LIN {X 0,Y 474.638,Z 146.861,A -85,B 0,C 180,E1 -7446.642,E2 -7446.642} C_VEL
LIN {X 0,Y 474.676,Z 147.003,A -85,B 0,C 180,E1 -7448.104,E2 -7448.104} C_VEL
LIN {X 0,Y 475.943,Z 154.468,A -85,B 0,C 180,E1 -7449.695,E2 -7449.695} C_VEL
LIN {X 0,Y 475.766,Z 161.873,A -85,B 0,C 180,E1 -7451.18,E2 -7451.18} C_VEL
LIN {X 0,Y 475.04,Z 165.15,A -85,B 0,C 180,E1 -7451.743,E2 -7451.743} C_VEL
LIN {X 0,Y 472.97,Z 170.29,A -85,B 0,C 180,E1 -7452.392,E2 -7452.392} C_VEL
LIN {X 0,Y 471.001,Z 176.225,A -85,B 0,C 180,E1 -7452.91,E2 -7452.91} C_VEL
LIN {X 0,Y 470.387,Z 181.246,A -85,B 0,C 180,E1 -7453.195,E2 -7453.195} C_VEL
LIN {X 0,Y 470.756,Z 184.775,A -85,B 0,C 180,E1 -7453.315,E2 -7453.315} C_VEL
LIN {X 0,Y 471.43,Z 190.109,A -85,B 0,C 180,E1 -7453.423,E2 -7453.423} C_VEL
LIN {X 0,Y 470.672,Z 280.468,A -85,B 0,C 180,E1 -7454.825,E2 -7454.825} C_VEL
LIN {X 0,Y 470.313,Z 294.355,A -85,B 0,C 180,E1 -7455.228,E2 -7455.228} C_VEL
LIN {X 0,Y 469.955,Z 306.775,A -85,B 0,C 180,E1 -7455.77,E2 -7455.77} C_VEL
LIN {X 0,Y 469.52,Z 318.965,A -85,B 0,C 180,E1 -7456.497,E2 -7456.497} C_VEL
LIN {X 0,Y 469.081,Z 330.013,A -85,B 0,C 180,E1 -7457.343,E2 -7457.343} C_VEL
LIN {X 0,Y 468.559,Z 340.263,A -85,B 0,C 180,E1 -7458.317,E2 -7458.317} C_VEL
LIN {X 0,Y 468.098,Z 349.46,A -85,B 0,C 180,E1 -7459.402,E2 -7459.402} C_VEL
LIN {X 0,Y 467.642,Z 358.386,A -85,B 0,C 180,E1 -7460.703,E2 -7460.703} C_VEL
LIN {X 0,Y 467.255,Z 365.574,A -85,B 0,C 180,E1 -7462.003,E2 -7462.003} C_VEL
LIN {X 0,Y 467.028,Z 371.353,A -85,B 0,C 180,E1 -7463.313,E2 -7463.313} C_VEL
LIN {X 0,Y 466.805,Z 376.452,A -85,B 0,C 180,E1 -7464.817,E2 -7464.817} C_VEL
LIN {X 0,Y 466.751,Z 378.743,A -85,B 0,C 180,E1 -7465.682,E2 -7465.682} C_VEL
LIN {X 0,Y 466.79,Z 380.605,A -85,B 0,C 180,E1 -7466.547,E2 -7466.547} C_VEL
LIN {X 0,Y 466.693,Z 382.013,A -85,B 0,C 180,E1 -7467.411,E2 -7467.411} C_VEL
LIN {X 0,Y 466.621,Z 383.629,A -85,B 0,C 180,E1 -7469.137,E2 -7469.137} C_VEL
LIN {X 0,Y 466.601,Z 383.866,A -85,B 0,C 180,E1 -7470,E2 -7470} C_VEL
LIN {X 0,Y 466.621,Z 383.68,A -85,B 0,C 180,E1 -7470.863,E2 -7470.863} C_VEL
LIN {X 0,Y 466.693,Z 382.129,A -85,B 0,C 180,E1 -7472.589,E2 -7472.589} C_VEL
LIN {X 0,Y 466.788,Z 380.771,A -85,B 0,C 180,E1 -7473.453,E2 -7473.453} C_VEL
LIN {X 0,Y 466.736,Z 377.908,A -85,B 0,C 180,E1 -7474.75,E2 -7474.75} C_VEL
LIN {X 0,Y 466.975,Z 374.018,A -85,B 0,C 180,E1 -7476.047,E2 -7476.047} C_VEL
LIN {X 0,Y 467.1,Z 369.005,A -85,B 0,C 180,E1 -7477.348,E2 -7477.348} C_VEL
LIN {X 0,Y 467.381,Z 362.693,A -85,B 0,C 180,E1 -7478.648,E2 -7478.648} C_VEL
LIN {X 0,Y 467.761,Z 354.79,A -85,B 0,C 180,E1 -7479.95,E2 -7479.95} C_VEL
LIN {X 0,Y 468.291,Z 344.958,A -85,B 0,C 180,E1 -7481.251,E2 -7481.251} C_VEL
LIN {X 0,Y 468.868,Z 334.644,A -85,B 0,C 180,E1 -7482.333,E2 -7482.333} C_VEL
LIN {X 0,Y 469.315,Z 323.077,A -85,B 0,C 180,E1 -7483.306,E2 -7483.306} C_VEL
LIN {X 0,Y 469.774,Z 311.433,A -85,B 0,C 180,E1 -7484.07,E2 -7484.07} C_VEL
LIN {X 0,Y 470.257,Z 299.391,A -85,B 0,C 180,E1 -7484.663,E2 -7484.663} C_VEL
LIN {X 0,Y 470.544,Z 286.28,A -85,B 0,C 180,E1 -7485.124,E2 -7485.124} C_VEL
LIN {X 0,Y 470.782,Z 273.664,A -85,B 0,C 180,E1 -7485.393,E2 -7485.393} C_VEL
LIN {X 0,Y 471.364,Z 188.194,A -85,B 0,C 180,E1 -7486.702,E2 -7486.702} C_VEL
LIN {X 0,Y 468.444,Z 172.801,A -85,B 0,C 180,E1 -7487.059,E2 -7487.059} C_VEL
LIN {X 0,Y 469,Z 157.256,A -85,B 0,C 180,E1 -7490.161,E2 -7490.161} C_VEL
LIN {X 0,Y 468.247,Z 151.065,A -85,B 0,C 180,E1 -7491.476,E2 -7491.476} C_VEL
LIN {X 0,Y 467.603,Z 147.741,A -85,B 0,C 180,E1 -7492.245,E2 -7492.245} C_VEL
LIN {X 0,Y 467.616,Z 147.734,A -85,B 0,C 180,E1 -7495.608,E2 -7495.608} C_VEL
LIN {X 0,Y 467.622,Z 147.732,A -85,B 0,C 180,E1 -7497.769,E2 -7497.769} C_VEL
LIN {X 0,Y 467.569,Z 147.741,A -85,B 0,C 180,E1 -7501.044,E2 -7501.044} C_VEL
LIN {X 0,Y 467.578,Z 147.741,A -85,B 0,C 180,E1 -7504.24,E2 -7504.24} C_VEL
LIN {X 0,Y 467.549,Z 147.741,A -85,B 0,C 180,E1 -7507.186,E2 -7507.186} C_VEL
LIN {X 0,Y 467.575,Z 147.745,A -85,B 0,C 180,E1 -7510.265,E2 -7510.265} C_VEL
LIN {X 0,Y 467.587,Z 147.74,A -85,B 0,C 180,E1 -7512.567,E2 -7512.567} C_VEL
LIN {X 0,Y 467.571,Z 147.738,A -85,B 0,C 180,E1 -7515.053,E2 -7515.053} C_VEL
LIN {X 0,Y 467.589,Z 147.736,A -85,B 0,C 180,E1 -7517.44,E2 -7517.44} C_VEL
LIN {X 0,Y 467.583,Z 147.737,A -85,B 0,C 180,E1 -7520.855,E2 -7520.855} C_VEL
LIN {X 0,Y 467.559,Z 147.743,A -85,B 0,C 180,E1 -7524.261,E2 -7524.261} C_VEL
LIN {X 0,Y 467.582,Z 147.739,A -85,B 0,C 180,E1 -7527.321,E2 -7527.321} C_VEL
LIN {X 0,Y 467.569,Z 147.738,A -85,B 0,C 180,E1 -7530.667,E2 -7530.667} C_VEL
LIN {X 0,Y 467.616,Z 147.735,A -85,B 0,C 180,E1 -7533.2,E2 -7533.2} C_VEL
LIN {X 0,Y 467.592,Z 147.735,A -85,B 0,C 180,E1 -7536.468,E2 -7536.468} C_VEL
LIN {X 0,Y 467.624,Z 147.735,A -85,B 0,C 180,E1 -7539.777,E2 -7539.777} C_VEL
LIN {X 0,Y 467.608,Z 147.733,A -85,B 0,C 180,E1 -7542.507,E2 -7542.507} C_VEL
LIN {X 0,Y 467.606,Z 147.741,A -85,B 0,C 180,E1 -7545.196,E2 -7545.196} C_VEL
LIN {X 0,Y 467.655,Z 147.728,A -85,B 0,C 180,E1 -7547.854,E2 -7547.854} C_VEL
LIN {X 0,Y 467.681,Z 147.729,A -85,B 0,C 180,E1 -7551.357,E2 -7551.357} C_VEL
LIN {X 0,Y 467.734,Z 147.718,A -85,B 0,C 180,E1 -7553.962,E2 -7553.962} C_VEL
LIN {X 0,Y 467.859,Z 147.704,A -85,B 0,C 180,E1 -7557.417,E2 -7557.417} C_VEL
LIN {X 0,Y 467.881,Z 147.699,A -85,B 0,C 180,E1 -7560,E2 -7560} C_VEL
LIN {X 0,Y 467.858,Z 147.708,A -85,B 0,C 180,E1 -7562.583,E2 -7562.583} C_VEL
LIN {X 0,Y 467.735,Z 147.719,A -85,B 0,C 180,E1 -7566.037,E2 -7566.037} C_VEL
LIN {X 0,Y 467.679,Z 147.731,A -85,B 0,C 180,E1 -7568.643,E2 -7568.643} C_VEL
LIN {X 0,Y 467.655,Z 147.731,A -85,B 0,C 180,E1 -7572.145,E2 -7572.145} C_VEL
LIN {X 0,Y 467.638,Z 147.731,A -85,B 0,C 180,E1 -7575.695,E2 -7575.695} C_VEL
LIN {X 0,Y 467.621,Z 147.732,A -85,B 0,C 180,E1 -7579.308,E2 -7579.308} C_VEL
LIN {X 0,Y 467.534,Z 147.75,A -85,B 0,C 180,E1 -7582.074,E2 -7582.074} C_VEL
LIN {X 0,Y 467.583,Z 147.737,A -85,B 0,C 180,E1 -7584.889,E2 -7584.889} C_VEL
LIN {X 0,Y 467.618,Z 147.737,A -85,B 0,C 180,E1 -7587.769,E2 -7587.769} C_VEL
LIN {X 0,Y 467.567,Z 147.739,A -85,B 0,C 180,E1 -7591.045,E2 -7591.045} C_VEL
LIN {X 0,Y 467.587,Z 147.738,A -85,B 0,C 180,E1 -7594.242,E2 -7594.242} C_VEL
LIN {X 0,Y 467.542,Z 147.744,A -85,B 0,C 180,E1 -7597.186,E2 -7597.186} C_VEL
LIN {X 0,Y 467.57,Z 147.739,A -85,B 0,C 180,E1 -7600.266,E2 -7600.266} C_VEL
LIN {X 0,Y 467.548,Z 147.745,A -85,B 0,C 180,E1 -7603.745,E2 -7603.745} C_VEL
LIN {X 0,Y 467.548,Z 147.741,A -85,B 0,C 180,E1 -7606.255,E2 -7606.255} C_VEL
LIN {X 0,Y 467.567,Z 147.74,A -85,B 0,C 180,E1 -7608.725,E2 -7608.725} C_VEL
LIN {X 0,Y 467.564,Z 147.739,A -85,B 0,C 180,E1 -7611.956,E2 -7611.956} C_VEL
LIN {X 0,Y 467.559,Z 147.747,A -85,B 0,C 180,E1 -7615.167,E2 -7615.167} C_VEL
LIN {X 0,Y 467.581,Z 147.737,A -85,B 0,C 180,E1 -7618.26,E2 -7618.26} C_VEL
LIN {X 0,Y 467.545,Z 147.745,A -85,B 0,C 180,E1 -7621.248,E2 -7621.248} C_VEL
LIN {X 0,Y 467.592,Z 147.743,A -85,B 0,C 180,E1 -7624.494,E2 -7624.494} C_VEL
LIN {X 0,Y 467.598,Z 147.812,A -85,B 0,C 180,E1 -7624.643,E2 -7624.643} C_VEL
LIN {X 0,Y 469.719,Z 159.111,A -85,B 0,C 180,E1 -7626.874,E2 -7626.874} C_VEL
LIN {X 0,Y 469.057,Z 174.117,A -85,B 0,C 180,E1 -7629.613,E2 -7629.613} C_VEL
LIN {X 0,Y 468.416,Z 190.342,A -85,B 0,C 180,E1 -7632.538,E2 -7632.538} C_VEL
LIN {X 0,Y 468.346,Z 192.794,A -85,B 0,C 180,E1 -7632.978,E2 -7632.978} C_VEL
LIN {X 0,Y 471.213,Z 210.729,A -85,B 0,C 180,E1 -7633.367,E2 -7633.367} C_VEL
LIN {X 0,Y 470.577,Z 300.893,A -85,B 0,C 180,E1 -7634.766,E2 -7634.766} C_VEL
LIN {X 0,Y 470.209,Z 314.155,A -85,B 0,C 180,E1 -7635.142,E2 -7635.142} C_VEL
LIN {X 0,Y 469.778,Z 326.312,A -85,B 0,C 180,E1 -7635.654,E2 -7635.654} C_VEL
LIN {X 0,Y 469.262,Z 338.578,A -85,B 0,C 180,E1 -7636.356,E2 -7636.356} C_VEL
LIN {X 0,Y 468.763,Z 350.191,A -85,B 0,C 180,E1 -7637.226,E2 -7637.226} C_VEL
LIN {X 0,Y 468.251,Z 360.609,A -85,B 0,C 180,E1 -7638.2,E2 -7638.2} C_VEL
LIN {X 0,Y 467.794,Z 369.142,A -85,B 0,C 180,E1 -7639.176,E2 -7639.176} C_VEL
LIN {X 0,Y 467.46,Z 377.017,A -85,B 0,C 180,E1 -7640.262,E2 -7640.262} C_VEL
LIN {X 0,Y 467.108,Z 384.706,A -85,B 0,C 180,E1 -7641.565,E2 -7641.565} C_VEL
LIN {X 0,Y 466.853,Z 391.796,A -85,B 0,C 180,E1 -7643.083,E2 -7643.083} C_VEL
LIN {X 0,Y 466.762,Z 396.513,A -85,B 0,C 180,E1 -7644.384,E2 -7644.384} C_VEL
LIN {X 0,Y 466.645,Z 400.115,A -85,B 0,C 180,E1 -7645.681,E2 -7645.681} C_VEL
LIN {X 0,Y 466.66,Z 401.975,A -85,B 0,C 180,E1 -7646.546,E2 -7646.546} C_VEL
LIN {X 0,Y 466.66,Z 403.369,A -85,B 0,C 180,E1 -7647.411,E2 -7647.411} C_VEL
LIN {X 0,Y 466.59,Z 404.969,A -85,B 0,C 180,E1 -7649.137,E2 -7649.137} C_VEL
LIN {X 0,Y 466.6,Z 405.185,A -85,B 0,C 180,E1 -7650,E2 -7650} C_VEL
LIN {X 0,Y 466.607,Z 404.363,A -85,B 0,C 180,E1 -7651.726,E2 -7651.726} C_VEL
LIN {X 0,Y 466.66,Z 403.37,A -85,B 0,C 180,E1 -7652.59,E2 -7652.59} C_VEL
LIN {X 0,Y 466.66,Z 401.976,A -85,B 0,C 180,E1 -7653.454,E2 -7653.454} C_VEL
LIN {X 0,Y 466.688,Z 399.044,A -85,B 0,C 180,E1 -7654.751,E2 -7654.751} C_VEL
LIN {X 0,Y 466.753,Z 395.074,A -85,B 0,C 180,E1 -7656.05,E2 -7656.05} C_VEL
LIN {X 0,Y 466.944,Z 388.971,A -85,B 0,C 180,E1 -7657.568,E2 -7657.568} C_VEL
LIN {X 0,Y 467.215,Z 382.3,A -85,B 0,C 180,E1 -7658.869,E2 -7658.869} C_VEL
LIN {X 0,Y 467.578,Z 374.024,A -85,B 0,C 180,E1 -7660.172,E2 -7660.172} C_VEL
LIN {X 0,Y 468.022,Z 365.541,A -85,B 0,C 180,E1 -7661.257,E2 -7661.257} C_VEL
LIN {X 0,Y 468.58,Z 355.481,A -85,B 0,C 180,E1 -7662.302,E2 -7662.302} C_VEL
LIN {X 0,Y 468.966,Z 344.686,A -85,B 0,C 180,E1 -7663.211,E2 -7663.211} C_VEL
LIN {X 0,Y 469.487,Z 333.316,A -85,B 0,C 180,E1 -7663.968,E2 -7663.968} C_VEL
LIN {X 0,Y 469.968,Z 321.649,A -85,B 0,C 180,E1 -7664.561,E2 -7664.561} C_VEL
LIN {X 0,Y 470.351,Z 310.034,A -85,B 0,C 180,E1 -7664.992,E2 -7664.992} C_VEL
LIN {X 0,Y 470.631,Z 296.424,A -85,B 0,C 180,E1 -7665.315,E2 -7665.315} C_VEL
LIN {X 0,Y 471.101,Z 210.051,A -85,B 0,C 180,E1 -7666.645,E2 -7666.645} C_VEL
LIN {X 0,Y 468.324,Z 192.816,A -85,B 0,C 180,E1 -7667.016,E2 -7667.016} C_VEL
LIN {X 0,Y 468.935,Z 176.595,A -85,B 0,C 180,E1 -7669.935,E2 -7669.935} C_VEL
LIN {X 0,Y 469.569,Z 162.843,A -85,B 0,C 180,E1 -7672.436,E2 -7672.436} C_VEL
LIN {X 0,Y 469.566,Z 157.831,A -85,B 0,C 180,E1 -7673.367,E2 -7673.367} C_VEL
LIN {X 0,Y 467.586,Z 147.743,A -85,B 0,C 180,E1 -7675.407,E2 -7675.407} C_VEL
LIN {X 0,Y 467.545,Z 147.743,A -85,B 0,C 180,E1 -7678.752,E2 -7678.752} C_VEL
LIN {X 0,Y 467.559,Z 147.74,A -85,B 0,C 180,E1 -7681.742,E2 -7681.742} C_VEL
LIN {X 0,Y 467.559,Z 147.747,A -85,B 0,C 180,E1 -7684.833,E2 -7684.833} C_VEL
LIN {X 0,Y 467.564,Z 147.739,A -85,B 0,C 180,E1 -7688.044,E2 -7688.044} C_VEL
LIN {X 0,Y 467.567,Z 147.739,A -85,B 0,C 180,E1 -7691.404,E2 -7691.404} C_VEL
LIN {X 0,Y 467.565,Z 147.742,A -85,B 0,C 180,E1 -7694.947,E2 -7694.947} C_VEL
LIN {X 0,Y 467.573,Z 147.744,A -85,B 0,C 180,E1 -7698.597,E2 -7698.597} C_VEL
LIN {X 0,Y 467.562,Z 147.742,A -85,B 0,C 180,E1 -7701.955,E2 -7701.955} C_VEL
LIN {X 0,Y 467.562,Z 147.739,A -85,B 0,C 180,E1 -7705.167,E2 -7705.167} C_VEL
LIN {X 0,Y 467.582,Z 147.744,A -85,B 0,C 180,E1 -7708.26,E2 -7708.26} C_VEL
LIN {X 0,Y 467.555,Z 147.74,A -85,B 0,C 180,E1 -7711.249,E2 -7711.249} C_VEL
LIN {X 0,Y 467.584,Z 147.742,A -85,B 0,C 180,E1 -7714.158,E2 -7714.158} C_VEL
LIN {X 0,Y 467.575,Z 147.737,A -85,B 0,C 180,E1 -7716.996,E2 -7716.996} C_VEL
LIN {X 0,Y 467.622,Z 147.739,A -85,B 0,C 180,E1 -7719.777,E2 -7719.777} C_VEL
LIN {X 0,Y 467.597,Z 147.735,A -85,B 0,C 180,E1 -7722.506,E2 -7722.506} C_VEL
LIN {X 0,Y 467.606,Z 147.736,A -85,B 0,C 180,E1 -7725.196,E2 -7725.196} C_VEL
LIN {X 0,Y 467.656,Z 147.732,A -85,B 0,C 180,E1 -7727.855,E2 -7727.855} C_VEL
LIN {X 0,Y 467.68,Z 147.731,A -85,B 0,C 180,E1 -7731.357,E2 -7731.357} C_VEL
LIN {X 0,Y 467.735,Z 147.719,A -85,B 0,C 180,E1 -7733.963,E2 -7733.963} C_VEL
LIN {X 0,Y 467.859,Z 147.709,A -85,B 0,C 180,E1 -7737.417,E2 -7737.417} C_VEL
LIN {X 0,Y 467.882,Z 147.7,A -85,B 0,C 180,E1 -7740,E2 -7740} C_VEL
LIN {X 0,Y 467.859,Z 147.703,A -85,B 0,C 180,E1 -7742.583,E2 -7742.583} C_VEL
LIN {X 0,Y 467.724,Z 147.719,A -85,B 0,C 180,E1 -7746.038,E2 -7746.038} C_VEL
LIN {X 0,Y 467.68,Z 147.728,A -85,B 0,C 180,E1 -7748.643,E2 -7748.643} C_VEL
LIN {X 0,Y 467.656,Z 147.728,A -85,B 0,C 180,E1 -7752.146,E2 -7752.146} C_VEL
LIN {X 0,Y 467.639,Z 147.729,A -85,B 0,C 180,E1 -7755.695,E2 -7755.695} C_VEL
LIN {X 0,Y 467.618,Z 147.739,A -85,B 0,C 180,E1 -7758.765,E2 -7758.765} C_VEL
LIN {X 0,Y 467.58,Z 147.738,A -85,B 0,C 180,E1 -7761.268,E2 -7761.268} C_VEL
LIN {X 0,Y 467.572,Z 147.739,A -85,B 0,C 180,E1 -7763.943,E2 -7763.943} C_VEL
LIN {X 0,Y 467.617,Z 147.735,A -85,B 0,C 180,E1 -7766.8,E2 -7766.8} C_VEL
LIN {X 0,Y 467.554,Z 147.741,A -85,B 0,C 180,E1 -7769.738,E2 -7769.738} C_VEL
LIN {X 0,Y 467.584,Z 147.738,A -85,B 0,C 180,E1 -7772.759,E2 -7772.759} C_VEL
LIN {X 0,Y 467.554,Z 147.744,A -85,B 0,C 180,E1 -7775.89,E2 -7775.89} C_VEL
LIN {X 0,Y 467.583,Z 147.736,A -85,B 0,C 180,E1 -7779.145,E2 -7779.145} C_VEL
LIN {X 0,Y 467.587,Z 147.737,A -85,B 0,C 180,E1 -7782.567,E2 -7782.567} C_VEL
LIN {X 0,Y 467.571,Z 147.738,A -85,B 0,C 180,E1 -7785.053,E2 -7785.053} C_VEL
LIN {X 0,Y 467.59,Z 147.739,A -85,B 0,C 180,E1 -7787.44,E2 -7787.44} C_VEL
LIN {X 0,Y 467.561,Z 147.739,A -85,B 0,C 180,E1 -7790.853,E2 -7790.853} C_VEL
LIN {X 0,Y 467.56,Z 147.74,A -85,B 0,C 180,E1 -7794.261,E2 -7794.261} C_VEL
LIN {X 0,Y 467.581,Z 147.742,A -85,B 0,C 180,E1 -7797.322,E2 -7797.322} C_VEL
LIN {X 0,Y 467.571,Z 147.738,A -85,B 0,C 180,E1 -7800.668,E2 -7800.668} C_VEL
LIN {X 0,Y 467.619,Z 147.738,A -85,B 0,C 180,E1 -7803.2,E2 -7803.2} C_VEL
LIN {X 0,Y 467.595,Z 147.738,A -85,B 0,C 180,E1 -7806.468,E2 -7806.468} C_VEL
LIN {X 0,Y 467.632,Z 147.918,A -85,B 0,C 180,E1 -7807.931,E2 -7807.931} C_VEL
LIN {X 0,Y 468.992,Z 155.682,A -85,B 0,C 180,E1 -7809.61,E2 -7809.61} C_VEL
LIN {X 0,Y 468.564,Z 169.167,A -85,B 0,C 180,E1 -7812.318,E2 -7812.318} C_VEL
LIN {X 0,Y 468.434,Z 172.751,A -85,B 0,C 180,E1 -7813.024,E2 -7813.024} C_VEL
LIN {X 0,Y 470.756,Z 184.775,A -85,B 0,C 180,E1 -7813.315,E2 -7813.315} C_VEL
LIN {X 0,Y 470.8,Z 187.997,A -85,B 0,C 180,E1 -7813.367,E2 -7813.367} C_VEL
LIN {X 0,Y 469.376,Z 192.433,A -85,B 0,C 180,E1 -7813.384,E2 -7813.384} C_VEL
LIN {X 0,Y 465.208,Z 201.121,A -85,B 0,C 180,E1 -7813.366,E2 -7813.366} C_VEL
LIN {X 0,Y 464.48,Z 205.116,A -85,B 0,C 180,E1 -7813.402,E2 -7813.402} C_VEL
LIN {X 0,Y 463.829,Z 280.648,A -85,B 0,C 180,E1 -7814.595,E2 -7814.595} C_VEL
LIN {X 0,Y 463.469,Z 294.528,A -85,B 0,C 180,E1 -7815.005,E2 -7815.005} C_VEL
LIN {X 0,Y 463.083,Z 306.945,A -85,B 0,C 180,E1 -7815.554,E2 -7815.554} C_VEL
LIN {X 0,Y 462.643,Z 318.812,A -85,B 0,C 180,E1 -7816.27,E2 -7816.27} C_VEL
LIN {X 0,Y 462.175,Z 328.894,A -85,B 0,C 180,E1 -7817.039,E2 -7817.039} C_VEL
LIN {X 0,Y 461.655,Z 339.368,A -85,B 0,C 180,E1 -7818.029,E2 -7818.029} C_VEL
LIN {X 0,Y 461.162,Z 347.927,A -85,B 0,C 180,E1 -7819.018,E2 -7819.018} C_VEL
LIN {X 0,Y 460.746,Z 355.81,A -85,B 0,C 180,E1 -7820.119,E2 -7820.119} C_VEL
LIN {X 0,Y 460.315,Z 363.517,A -85,B 0,C 180,E1 -7821.439,E2 -7821.439} C_VEL
LIN {X 0,Y 460.001,Z 370.587,A -85,B 0,C 180,E1 -7822.979,E2 -7822.979} C_VEL
LIN {X 0,Y 459.87,Z 375.297,A -85,B 0,C 180,E1 -7824.299,E2 -7824.299} C_VEL
LIN {X 0,Y 459.658,Z 378.906,A -85,B 0,C 180,E1 -7825.616,E2 -7825.616} C_VEL
LIN {X 0,Y 459.701,Z 380.769,A -85,B 0,C 180,E1 -7826.494,E2 -7826.494} C_VEL
LIN {X 0,Y 459.617,Z 382.175,A -85,B 0,C 180,E1 -7827.371,E2 -7827.371} C_VEL
LIN {X 0,Y 459.525,Z 383.792,A -85,B 0,C 180,E1 -7829.124,E2 -7829.124} C_VEL
LIN {X 0,Y 459.504,Z 384.028,A -85,B 0,C 180,E1 -7830,E2 -7830} C_VEL
LIN {X 0,Y 459.525,Z 383.841,A -85,B 0,C 180,E1 -7830.876,E2 -7830.876} C_VEL
LIN {X 0,Y 459.617,Z 382.29,A -85,B 0,C 180,E1 -7832.629,E2 -7832.629} C_VEL
LIN {X 0,Y 459.699,Z 380.933,A -85,B 0,C 180,E1 -7833.506,E2 -7833.506} C_VEL
LIN {X 0,Y 459.664,Z 378.069,A -85,B 0,C 180,E1 -7834.824,E2 -7834.824} C_VEL
LIN {X 0,Y 459.912,Z 374.179,A -85,B 0,C 180,E1 -7836.141,E2 -7836.141} C_VEL
LIN {X 0,Y 460.05,Z 369.165,A -85,B 0,C 180,E1 -7837.461,E2 -7837.461} C_VEL
LIN {X 0,Y 460.361,Z 362.853,A -85,B 0,C 180,E1 -7838.781,E2 -7838.781} C_VEL
LIN {X 0,Y 460.744,Z 354.95,A -85,B 0,C 180,E1 -7840.103,E2 -7840.103} C_VEL
LIN {X 0,Y 461.34,Z 345.116,A -85,B 0,C 180,E1 -7841.422,E2 -7841.422} C_VEL
LIN {X 0,Y 461.93,Z 334.801,A -85,B 0,C 180,E1 -7842.521,E2 -7842.521} C_VEL
LIN {X 0,Y 462.382,Z 323.681,A -85,B 0,C 180,E1 -7843.474,E2 -7843.474} C_VEL
LIN {X 0,Y 462.908,Z 311.587,A -85,B 0,C 180,E1 -7844.283,E2 -7844.283} C_VEL
LIN {X 0,Y 463.387,Z 299.543,A -85,B 0,C 180,E1 -7844.885,E2 -7844.885} C_VEL
LIN {X 0,Y 463.694,Z 286.428,A -85,B 0,C 180,E1 -7845.353,E2 -7845.353} C_VEL
LIN {X 0,Y 463.943,Z 273.798,A -85,B 0,C 180,E1 -7845.626,E2 -7845.626} C_VEL
LIN {X 0,Y 464.469,Z 188.389,A -85,B 0,C 180,E1 -7846.956,E2 -7846.956} C_VEL
LIN {X 0,Y 461.514,Z 172.908,A -85,B 0,C 180,E1 -7847.332,E2 -7847.332} C_VEL
LIN {X 0,Y 462.052,Z 158.489,A -85,B 0,C 180,E1 -7850.245,E2 -7850.245} C_VEL
LIN {X 0,Y 461.404,Z 152.909,A -85,B 0,C 180,E1 -7851.442,E2 -7851.442} C_VEL
LIN {X 0,Y 460.568,Z 148.617,A -85,B 0,C 180,E1 -7852.426,E2 -7852.426} C_VEL
LIN {X 0,Y 460.57,Z 148.612,A -85,B 0,C 180,E1 -7855.802,E2 -7855.802} C_VEL
LIN {X 0,Y 460.554,Z 148.614,A -85,B 0,C 180,E1 -7858.233,E2 -7858.233} C_VEL
LIN {X 0,Y 460.522,Z 148.617,A -85,B 0,C 180,E1 -7861.282,E2 -7861.282} C_VEL
LIN {X 0,Y 460.524,Z 148.624,A -85,B 0,C 180,E1 -7864.504,E2 -7864.504} C_VEL
LIN {X 0,Y 460.502,Z 148.619,A -85,B 0,C 180,E1 -7867.623,E2 -7867.623} C_VEL
LIN {X 0,Y 460.54,Z 148.621,A -85,B 0,C 180,E1 -7870.269,E2 -7870.269} C_VEL
LIN {X 0,Y 460.501,Z 148.619,A -85,B 0,C 180,E1 -7873.375,E2 -7873.375} C_VEL
LIN {X 0,Y 460.5,Z 148.621,A -85,B 0,C 180,E1 -7876.624,E2 -7876.624} C_VEL
LIN {X 0,Y 460.542,Z 148.617,A -85,B 0,C 180,E1 -7879.73,E2 -7879.73} C_VEL
LIN {X 0,Y 460.5,Z 148.62,A -85,B 0,C 180,E1 -7882.524,E2 -7882.524} C_VEL
LIN {X 0,Y 460.546,Z 148.618,A -85,B 0,C 180,E1 -7885.624,E2 -7885.624} C_VEL
LIN {X 0,Y 460.537,Z 148.614,A -85,B 0,C 180,E1 -7888.744,E2 -7888.744} C_VEL
LIN {X 0,Y 460.581,Z 148.61,A -85,B 0,C 180,E1 -7892.254,E2 -7892.254} C_VEL
LIN {X 0,Y 460.558,Z 148.612,A -85,B 0,C 180,E1 -7894.705,E2 -7894.705} C_VEL
LIN {X 0,Y 460.51,Z 148.625,A -85,B 0,C 180,E1 -7897.571,E2 -7897.571} C_VEL
LIN {X 0,Y 460.569,Z 148.61,A -85,B 0,C 180,E1 -7900.384,E2 -7900.384} C_VEL
LIN {X 0,Y 460.565,Z 148.616,A -85,B 0,C 180,E1 -7903.146,E2 -7903.146} C_VEL
LIN {X 0,Y 460.554,Z 148.613,A -85,B 0,C 180,E1 -7905.868,E2 -7905.868} C_VEL
LIN {X 0,Y 460.611,Z 148.606,A -85,B 0,C 180,E1 -7908.559,E2 -7908.559} C_VEL
LIN {X 0,Y 460.694,Z 148.595,A -85,B 0,C 180,E1 -7912.108,E2 -7912.108} C_VEL
LIN {X 0,Y 460.693,Z 148.6,A -85,B 0,C 180,E1 -7914.748,E2 -7914.748} C_VEL
LIN {X 0,Y 460.824,Z 148.581,A -85,B 0,C 180,E1 -7917.378,E2 -7917.378} C_VEL
LIN {X 0,Y 460.852,Z 148.575,A -85,B 0,C 180,E1 -7920,E2 -7920} C_VEL
LIN {X 0,Y 460.823,Z 148.585,A -85,B 0,C 180,E1 -7922.622,E2 -7922.622} C_VEL
LIN {X 0,Y 460.701,Z 148.596,A -85,B 0,C 180,E1 -7926.13,E2 -7926.13} C_VEL
LIN {X 0,Y 460.626,Z 148.608,A -85,B 0,C 180,E1 -7928.776,E2 -7928.776} C_VEL
LIN {X 0,Y 460.612,Z 148.613,A -85,B 0,C 180,E1 -7932.445,E2 -7932.445} C_VEL
LIN {X 0,Y 460.599,Z 148.61,A -85,B 0,C 180,E1 -7935.998,E2 -7935.998} C_VEL
LIN {X 0,Y 460.567,Z 148.612,A -85,B 0,C 180,E1 -7939.616,E2 -7939.616} C_VEL
LIN {X 0,Y 460.51,Z 148.622,A -85,B 0,C 180,E1 -7942.429,E2 -7942.429} C_VEL
LIN {X 0,Y 460.552,Z 148.617,A -85,B 0,C 180,E1 -7945.798,E2 -7945.798} C_VEL
LIN {X 0,Y 460.55,Z 148.617,A -85,B 0,C 180,E1 -7948.233,E2 -7948.233} C_VEL
LIN {X 0,Y 460.52,Z 148.618,A -85,B 0,C 180,E1 -7951.283,E2 -7951.283} C_VEL
LIN {X 0,Y 460.53,Z 148.616,A -85,B 0,C 180,E1 -7954.505,E2 -7954.505} C_VEL
LIN {X 0,Y 460.498,Z 148.626,A -85,B 0,C 180,E1 -7957.624,E2 -7957.624} C_VEL
LIN {X 0,Y 460.534,Z 148.615,A -85,B 0,C 180,E1 -7960.269,E2 -7960.269} C_VEL
LIN {X 0,Y 460.508,Z 148.624,A -85,B 0,C 180,E1 -7963.375,E2 -7963.375} C_VEL
LIN {X 0,Y 460.508,Z 148.618,A -85,B 0,C 180,E1 -7966.626,E2 -7966.626} C_VEL
LIN {X 0,Y 460.525,Z 148.618,A -85,B 0,C 180,E1 -7969.733,E2 -7969.733} C_VEL
LIN {X 0,Y 460.499,Z 148.62,A -85,B 0,C 180,E1 -7972.524,E2 -7972.524} C_VEL
LIN {X 0,Y 460.537,Z 148.616,A -85,B 0,C 180,E1 -7975.623,E2 -7975.623} C_VEL
LIN {X 0,Y 460.538,Z 148.618,A -85,B 0,C 180,E1 -7978.745,E2 -7978.745} C_VEL
LIN {X 0,Y 460.532,Z 148.617,A -85,B 0,C 180,E1 -7982.266,E2 -7982.266} C_VEL
LIN {X 0,Y 460.552,Z 148.697,A -85,B 0,C 180,E1 -7984.43,E2 -7984.43} C_VEL
LIN {X 0,Y 462.756,Z 160.202,A -85,B 0,C 180,E1 -7986.742,E2 -7986.742} C_VEL
LIN {X 0,Y 462.085,Z 175.205,A -85,B 0,C 180,E1 -7989.524,E2 -7989.524} C_VEL
LIN {X 0,Y 461.472,Z 190.18,A -85,B 0,C 180,E1 -7992.267,E2 -7992.267} C_VEL
LIN {X 0,Y 461.348,Z 192.63,A -85,B 0,C 180,E1 -7992.712,E2 -7992.712} C_VEL
LIN {X 0,Y 464.446,Z 211.735,A -85,B 0,C 180,E1 -7993.136,E2 -7993.136} C_VEL
LIN {X 0,Y 463.749,Z 300.742,A -85,B 0,C 180,E1 -7994.536,E2 -7994.536} C_VEL
LIN {X 0,Y 463.348,Z 314,A -85,B 0,C 180,E1 -7994.917,E2 -7994.917} C_VEL
LIN {X 0,Y 462.903,Z 326.156,A -85,B 0,C 180,E1 -7995.436,E2 -7995.436} C_VEL
LIN {X 0,Y 462.348,Z 338.419,A -85,B 0,C 180,E1 -7996.148,E2 -7996.148} C_VEL
LIN {X 0,Y 461.773,Z 350.03,A -85,B 0,C 180,E1 -7997.029,E2 -7997.029} C_VEL
LIN {X 0,Y 461.287,Z 360.449,A -85,B 0,C 180,E1 -7998.019,E2 -7998.019} C_VEL
LIN {X 0,Y 460.799,Z 368.981,A -85,B 0,C 180,E1 -7999.01,E2 -7999.01} C_VEL
LIN {X 0,Y 460.449,Z 376.856,A -85,B 0,C 180,E1 -8000.113,E2 -8000.113} C_VEL
LIN {X 0,Y 460.045,Z 384.544,A -85,B 0,C 180,E1 -8001.434,E2 -8001.434} C_VEL
LIN {X 0,Y 459.772,Z 391.634,A -85,B 0,C 180,E1 -8002.976,E2 -8002.976} C_VEL
LIN {X 0,Y 459.661,Z 396.351,A -85,B 0,C 180,E1 -8004.296,E2 -8004.296} C_VEL
LIN {X 0,Y 459.563,Z 399.954,A -85,B 0,C 180,E1 -8005.615,E2 -8005.615} C_VEL
LIN {X 0,Y 459.557,Z 401.813,A -85,B 0,C 180,E1 -8006.493,E2 -8006.493} C_VEL
LIN {X 0,Y 459.581,Z 403.207,A -85,B 0,C 180,E1 -8007.371,E2 -8007.371} C_VEL
LIN {X 0,Y 459.495,Z 404.807,A -85,B 0,C 180,E1 -8009.124,E2 -8009.124} C_VEL
LIN {X 0,Y 459.503,Z 405.023,A -85,B 0,C 180,E1 -8010,E2 -8010} C_VEL
LIN {X 0,Y 459.52,Z 404.201,A -85,B 0,C 180,E1 -8011.753,E2 -8011.753} C_VEL
LIN {X 0,Y 459.581,Z 403.208,A -85,B 0,C 180,E1 -8012.629,E2 -8012.629} C_VEL
LIN {X 0,Y 459.557,Z 401.813,A -85,B 0,C 180,E1 -8013.507,E2 -8013.507} C_VEL
LIN {X 0,Y 459.616,Z 398.881,A -85,B 0,C 180,E1 -8014.824,E2 -8014.824} C_VEL
LIN {X 0,Y 459.714,Z 393.882,A -85,B 0,C 180,E1 -8016.431,E2 -8016.431} C_VEL
LIN {X 0,Y 459.902,Z 387.795,A -85,B 0,C 180,E1 -8017.905,E2 -8017.905} C_VEL
LIN {X 0,Y 460.213,Z 380.9,A -85,B 0,C 180,E1 -8019.227,E2 -8019.227} C_VEL
LIN {X 0,Y 460.555,Z 373.859,A -85,B 0,C 180,E1 -8020.329,E2 -8020.329} C_VEL
LIN {X 0,Y 461.04,Z 365.377,A -85,B 0,C 180,E1 -8021.43,E2 -8021.43} C_VEL
LIN {X 0,Y 461.612,Z 355.527,A -85,B 0,C 180,E1 -8022.47,E2 -8022.47} C_VEL
LIN {X 0,Y 461.965,Z 345.948,A -85,B 0,C 180,E1 -8023.303,E2 -8023.303} C_VEL
LIN {X 0,Y 462.505,Z 334.919,A -85,B 0,C 180,E1 -8024.071,E2 -8024.071} C_VEL
LIN {X 0,Y 463.022,Z 322.694,A -85,B 0,C 180,E1 -8024.729,E2 -8024.729} C_VEL
LIN {X 0,Y 463.483,Z 310.778,A -85,B 0,C 180,E1 -8025.191,E2 -8025.191} C_VEL
LIN {X 0,Y 463.775,Z 297.753,A -85,B 0,C 180,E1 -8025.519,E2 -8025.519} C_VEL
LIN {X 0,Y 464.408,Z 211.65,A -85,B 0,C 180,E1 -8026.863,E2 -8026.863} C_VEL
LIN {X 0,Y 461.371,Z 192.61,A -85,B 0,C 180,E1 -8027.288,E2 -8027.288} C_VEL
LIN {X 0,Y 462.031,Z 176.431,A -85,B 0,C 180,E1 -8030.246,E2 -8030.246} C_VEL
LIN {X 0,Y 462.67,Z 162.68,A -85,B 0,C 180,E1 -8032.79,E2 -8032.79} C_VEL
LIN {X 0,Y 462.584,Z 159.011,A -85,B 0,C 180,E1 -8033.486,E2 -8033.486} C_VEL
LIN {X 0,Y 460.544,Z 148.62,A -85,B 0,C 180,E1 -8035.61,E2 -8035.61} C_VEL
LIN {X 0,Y 460.508,Z 148.617,A -85,B 0,C 180,E1 -8038.236,E2 -8038.236} C_VEL
LIN {X 0,Y 460.521,Z 148.62,A -85,B 0,C 180,E1 -8041.282,E2 -8041.282} C_VEL
LIN {X 0,Y 460.524,Z 148.619,A -85,B 0,C 180,E1 -8044.504,E2 -8044.504} C_VEL
LIN {X 0,Y 460.501,Z 148.619,A -85,B 0,C 180,E1 -8047.623,E2 -8047.623} C_VEL
LIN {X 0,Y 460.525,Z 148.618,A -85,B 0,C 180,E1 -8050.267,E2 -8050.267} C_VEL
LIN {X 0,Y 460.508,Z 148.618,A -85,B 0,C 180,E1 -8053.374,E2 -8053.374} C_VEL
LIN {X 0,Y 460.508,Z 148.624,A -85,B 0,C 180,E1 -8056.625,E2 -8056.625} C_VEL
LIN {X 0,Y 460.535,Z 148.615,A -85,B 0,C 180,E1 -8059.731,E2 -8059.731} C_VEL
LIN {X 0,Y 460.497,Z 148.625,A -85,B 0,C 180,E1 -8062.524,E2 -8062.524} C_VEL
LIN {X 0,Y 460.545,Z 148.614,A -85,B 0,C 180,E1 -8065.624,E2 -8065.624} C_VEL
LIN {X 0,Y 460.537,Z 148.616,A -85,B 0,C 180,E1 -8068.744,E2 -8068.744} C_VEL
LIN {X 0,Y 460.55,Z 148.618,A -85,B 0,C 180,E1 -8072.261,E2 -8072.261} C_VEL
LIN {X 0,Y 460.539,Z 148.614,A -85,B 0,C 180,E1 -8074.704,E2 -8074.704} C_VEL
LIN {X 0,Y 460.51,Z 148.621,A -85,B 0,C 180,E1 -8077.571,E2 -8077.571} C_VEL
LIN {X 0,Y 460.567,Z 148.612,A -85,B 0,C 180,E1 -8080.384,E2 -8080.384} C_VEL
LIN {X 0,Y 460.604,Z 148.609,A -85,B 0,C 180,E1 -8084.059,E2 -8084.059} C_VEL
LIN {X 0,Y 460.609,Z 148.612,A -85,B 0,C 180,E1 -8087.666,E2 -8087.666} C_VEL
LIN {X 0,Y 460.627,Z 148.607,A -85,B 0,C 180,E1 -8091.224,E2 -8091.224} C_VEL
LIN {X 0,Y 460.701,Z 148.596,A -85,B 0,C 180,E1 -8093.87,E2 -8093.87} C_VEL
LIN {X 0,Y 460.823,Z 148.586,A -85,B 0,C 180,E1 -8097.378,E2 -8097.378} C_VEL
LIN {X 0,Y 460.852,Z 148.575,A -85,B 0,C 180,E1 -8100,E2 -8100} C_VEL
LIN {X 0,Y 460.824,Z 148.58,A -85,B 0,C 180,E1 -8102.622,E2 -8102.622} C_VEL
LIN {X 0,Y 460.688,Z 148.595,A -85,B 0,C 180,E1 -8106.13,E2 -8106.13} C_VEL
LIN {X 0,Y 460.627,Z 148.608,A -85,B 0,C 180,E1 -8108.776,E2 -8108.776} C_VEL
LIN {X 0,Y 460.613,Z 148.607,A -85,B 0,C 180,E1 -8112.445,E2 -8112.445} C_VEL
LIN {X 0,Y 460.6,Z 148.607,A -85,B 0,C 180,E1 -8115.998,E2 -8115.998} C_VEL
LIN {X 0,Y 460.571,Z 148.615,A -85,B 0,C 180,E1 -8118.902,E2 -8118.902} C_VEL
LIN {X 0,Y 460.516,Z 148.617,A -85,B 0,C 180,E1 -8121.486,E2 -8121.486} C_VEL
LIN {X 0,Y 460.542,Z 148.619,A -85,B 0,C 180,E1 -8124.332,E2 -8124.332} C_VEL
LIN {X 0,Y 460.573,Z 148.61,A -85,B 0,C 180,E1 -8127.244,E2 -8127.244} C_VEL
LIN {X 0,Y 460.511,Z 148.624,A -85,B 0,C 180,E1 -8130.24,E2 -8130.24} C_VEL
LIN {X 0,Y 460.529,Z 148.615,A -85,B 0,C 180,E1 -8133.325,E2 -8133.325} C_VEL
LIN {X 0,Y 460.477,Z 148.625,A -85,B 0,C 180,E1 -8136.53,E2 -8136.53} C_VEL
LIN {X 0,Y 460.533,Z 148.62,A -85,B 0,C 180,E1 -8139.863,E2 -8139.863} C_VEL
LIN {X 0,Y 460.514,Z 148.617,A -85,B 0,C 180,E1 -8142.901,E2 -8142.901} C_VEL
LIN {X 0,Y 460.513,Z 148.625,A -85,B 0,C 180,E1 -8145.831,E2 -8145.831} C_VEL
LIN {X 0,Y 460.532,Z 148.615,A -85,B 0,C 180,E1 -8148.989,E2 -8148.989} C_VEL
LIN {X 0,Y 460.52,Z 148.619,A -85,B 0,C 180,E1 -8151.266,E2 -8151.266} C_VEL
LIN {X 0,Y 460.51,Z 148.618,A -85,B 0,C 180,E1 -8154.554,E2 -8154.554} C_VEL
LIN {X 0,Y 460.531,Z 148.62,A -85,B 0,C 180,E1 -8157.716,E2 -8157.716} C_VEL
LIN {X 0,Y 460.541,Z 148.615,A -85,B 0,C 180,E1 -8160.769,E2 -8160.769} C_VEL
LIN {X 0,Y 460.566,Z 148.616,A -85,B 0,C 180,E1 -8163.735,E2 -8163.735} C_VEL
LIN {X 0,Y 460.549,Z 148.616,A -85,B 0,C 180,E1 -8166.624,E2 -8166.624} C_VEL
LIN {X 0,Y 460.589,Z 148.814,A -85,B 0,C 180,E1 -8167.748,E2 -8167.748} C_VEL
LIN {X 0,Y 462.021,Z 156.911,A -85,B 0,C 180,E1 -8169.521,E2 -8169.521} C_VEL
LIN {X 0,Y 461.64,Z 169.313,A -85,B 0,C 180,E1 -8172.044,E2 -8172.044} C_VEL
LIN {X 0,Y 461.473,Z 173.035,A -85,B 0,C 180,E1 -8172.778,E2 -8172.778} C_VEL
LIN {X 0,Y 464.631,Z 190.299,A -85,B 0,C 180,E1 -8173.173,E2 -8173.173} C_VEL
LIN {X 0,Y 464.48,Z 205.116,A -85,B 0,C 180,E1 -8173.402,E2 -8173.402} C_VEL
LIN {X 0,Y 463.807,Z 210.969,A -85,B 0,C 180,E1 -8173.47,E2 -8173.47} C_VEL
LIN {X 0,Y 458.036,Z 229.97,A -85,B 0,C 180,E1 -8173.558,E2 -8173.558} C_VEL
LIN {X 0,Y 457.464,Z 235.815,A -85,B 0,C 180,E1 -8173.63,E2 -8173.63} C_VEL
LIN {X 0,Y 457.016,Z 280.827,A -85,B 0,C 180,E1 -8174.36,E2 -8174.36} C_VEL
LIN {X 0,Y 456.643,Z 294.702,A -85,B 0,C 180,E1 -8174.776,E2 -8174.776} C_VEL
LIN {X 0,Y 456.215,Z 307.115,A -85,B 0,C 180,E1 -8175.332,E2 -8175.332} C_VEL
LIN {X 0,Y 455.734,Z 318.981,A -85,B 0,C 180,E1 -8176.057,E2 -8176.057} C_VEL
LIN {X 0,Y 455.241,Z 329.185,A -85,B 0,C 180,E1 -8176.849,E2 -8176.849} C_VEL
LIN {X 0,Y 454.723,Z 339.534,A -85,B 0,C 180,E1 -8177.844,E2 -8177.844} C_VEL
LIN {X 0,Y 454.193,Z 348.093,A -85,B 0,C 180,E1 -8178.848,E2 -8178.848} C_VEL
LIN {X 0,Y 453.734,Z 355.975,A -85,B 0,C 180,E1 -8179.965,E2 -8179.965} C_VEL
LIN {X 0,Y 453.296,Z 363.682,A -85,B 0,C 180,E1 -8181.305,E2 -8181.305} C_VEL
LIN {X 0,Y 452.949,Z 370.751,A -85,B 0,C 180,E1 -8182.87,E2 -8182.87} C_VEL
LIN {X 0,Y 452.798,Z 375.46,A -85,B 0,C 180,E1 -8184.21,E2 -8184.21} C_VEL
LIN {X 0,Y 452.571,Z 379.07,A -85,B 0,C 180,E1 -8185.547,E2 -8185.547} C_VEL
LIN {X 0,Y 452.616,Z 380.932,A -85,B 0,C 180,E1 -8186.439,E2 -8186.439} C_VEL
LIN {X 0,Y 452.543,Z 382.338,A -85,B 0,C 180,E1 -8187.33,E2 -8187.33} C_VEL
LIN {X 0,Y 452.432,Z 383.954,A -85,B 0,C 180,E1 -8189.11,E2 -8189.11} C_VEL
LIN {X 0,Y 452.41,Z 384.19,A -85,B 0,C 180,E1 -8190,E2 -8190} C_VEL
LIN {X 0,Y 452.432,Z 384.003,A -85,B 0,C 180,E1 -8190.89,E2 -8190.89} C_VEL
LIN {X 0,Y 452.543,Z 382.451,A -85,B 0,C 180,E1 -8192.67,E2 -8192.67} C_VEL
LIN {X 0,Y 452.613,Z 381.094,A -85,B 0,C 180,E1 -8193.561,E2 -8193.561} C_VEL
LIN {X 0,Y 452.598,Z 378.23,A -85,B 0,C 180,E1 -8194.899,E2 -8194.899} C_VEL
LIN {X 0,Y 452.845,Z 374.34,A -85,B 0,C 180,E1 -8196.237,E2 -8196.237} C_VEL
LIN {X 0,Y 452.993,Z 369.326,A -85,B 0,C 180,E1 -8197.578,E2 -8197.578} C_VEL
LIN {X 0,Y 453.345,Z 363.013,A -85,B 0,C 180,E1 -8198.918,E2 -8198.918} C_VEL
LIN {X 0,Y 453.752,Z 355.109,A -85,B 0,C 180,E1 -8200.26,E2 -8200.26} C_VEL
LIN {X 0,Y 454.232,Z 347.052,A -85,B 0,C 180,E1 -8201.377,E2 -8201.377} C_VEL
LIN {X 0,Y 454.855,Z 337.217,A -85,B 0,C 180,E1 -8202.493,E2 -8202.493} C_VEL
LIN {X 0,Y 455.315,Z 327.546,A -85,B 0,C 180,E1 -8203.387,E2 -8203.387} C_VEL
LIN {X 0,Y 455.834,Z 317.086,A -85,B 0,C 180,E1 -8204.167,E2 -8204.167} C_VEL
LIN {X 0,Y 456.29,Z 305.613,A -85,B 0,C 180,E1 -8204.837,E2 -8204.837} C_VEL
LIN {X 0,Y 456.753,Z 292.643,A -85,B 0,C 180,E1 -8205.392,E2 -8205.392} C_VEL
LIN {X 0,Y 457.03,Z 279.986,A -85,B 0,C 180,E1 -8205.754,E2 -8205.754} C_VEL
LIN {X 0,Y 457.75,Z 189.661,A -85,B 0,C 180,E1 -8207.195,E2 -8207.195} C_VEL
LIN {X 0,Y 454.584,Z 173.119,A -85,B 0,C 180,E1 -8207.593,E2 -8207.593} C_VEL
LIN {X 0,Y 455.106,Z 158.605,A -85,B 0,C 180,E1 -8210.568,E2 -8210.568} C_VEL
LIN {X 0,Y 453.526,Z 149.495,A -85,B 0,C 180,E1 -8212.613,E2 -8212.613} C_VEL
LIN {X 0,Y 453.52,Z 149.491,A -85,B 0,C 180,E1 -8215.999,E2 -8215.999} C_VEL
LIN {X 0,Y 453.511,Z 149.497,A -85,B 0,C 180,E1 -8218.712,E2 -8218.712} C_VEL
LIN {X 0,Y 453.464,Z 149.496,A -85,B 0,C 180,E1 -8221.799,E2 -8221.799} C_VEL
LIN {X 0,Y 453.477,Z 149.496,A -85,B 0,C 180,E1 -8224.989,E2 -8224.989} C_VEL
LIN {X 0,Y 453.461,Z 149.502,A -85,B 0,C 180,E1 -8228.312,E2 -8228.312} C_VEL
LIN {X 0,Y 453.494,Z 149.496,A -85,B 0,C 180,E1 -8230.609,E2 -8230.609} C_VEL
LIN {X 0,Y 453.456,Z 149.496,A -85,B 0,C 180,E1 -8233.244,E2 -8233.244} C_VEL
LIN {X 0,Y 453.467,Z 149.498,A -85,B 0,C 180,E1 -8235.779,E2 -8235.779} C_VEL
LIN {X 0,Y 453.48,Z 149.5,A -85,B 0,C 180,E1 -8238.209,E2 -8238.209} C_VEL
LIN {X 0,Y 453.495,Z 149.492,A -85,B 0,C 180,E1 -8240.793,E2 -8240.793} C_VEL
LIN {X 0,Y 453.454,Z 149.504,A -85,B 0,C 180,E1 -8243.917,E2 -8243.917} C_VEL
LIN {X 0,Y 453.483,Z 149.494,A -85,B 0,C 180,E1 -8247.151,E2 -8247.151} C_VEL
LIN {X 0,Y 453.474,Z 149.496,A -85,B 0,C 180,E1 -8250.268,E2 -8250.268} C_VEL
LIN {X 0,Y 453.506,Z 149.494,A -85,B 0,C 180,E1 -8253.294,E2 -8253.294} C_VEL
LIN {X 0,Y 453.502,Z 149.491,A -85,B 0,C 180,E1 -8256.239,E2 -8256.239} C_VEL
LIN {X 0,Y 453.483,Z 149.496,A -85,B 0,C 180,E1 -8259.118,E2 -8259.118} C_VEL
LIN {X 0,Y 453.511,Z 149.491,A -85,B 0,C 180,E1 -8261.944,E2 -8261.944} C_VEL
LIN {X 0,Y 453.539,Z 149.487,A -85,B 0,C 180,E1 -8264.726,E2 -8264.726} C_VEL
LIN {X 0,Y 453.559,Z 149.484,A -85,B 0,C 180,E1 -8268.379,E2 -8268.379} C_VEL
LIN {X 0,Y 453.651,Z 149.472,A -85,B 0,C 180,E1 -8271.985,E2 -8271.985} C_VEL
LIN {X 0,Y 453.667,Z 149.474,A -85,B 0,C 180,E1 -8274.667,E2 -8274.667} C_VEL
LIN {X 0,Y 453.764,Z 149.46,A -85,B 0,C 180,E1 -8277.337,E2 -8277.337} C_VEL
LIN {X 0,Y 453.822,Z 149.451,A -85,B 0,C 180,E1 -8280,E2 -8280} C_VEL
LIN {X 0,Y 453.763,Z 149.465,A -85,B 0,C 180,E1 -8282.663,E2 -8282.663} C_VEL
LIN {X 0,Y 453.669,Z 149.473,A -85,B 0,C 180,E1 -8286.225,E2 -8286.225} C_VEL
LIN {X 0,Y 453.59,Z 149.483,A -85,B 0,C 180,E1 -8288.913,E2 -8288.913} C_VEL
LIN {X 0,Y 453.563,Z 149.49,A -85,B 0,C 180,E1 -8292.529,E2 -8292.529} C_VEL
LIN {X 0,Y 453.543,Z 149.492,A -85,B 0,C 180,E1 -8296.196,E2 -8296.196} C_VEL
LIN {X 0,Y 453.516,Z 149.489,A -85,B 0,C 180,E1 -8299.04,E2 -8299.04} C_VEL
LIN {X 0,Y 453.475,Z 149.498,A -85,B 0,C 180,E1 -8301.836,E2 -8301.836} C_VEL
LIN {X 0,Y 453.499,Z 149.492,A -85,B 0,C 180,E1 -8304.735,E2 -8304.735} C_VEL
LIN {X 0,Y 453.53,Z 149.495,A -85,B 0,C 180,E1 -8307.959,E2 -8307.959} C_VEL
LIN {X 0,Y 453.465,Z 149.499,A -85,B 0,C 180,E1 -8311.525,E2 -8311.525} C_VEL
LIN {X 0,Y 453.486,Z 149.493,A -85,B 0,C 180,E1 -8314.777,E2 -8314.777} C_VEL
LIN {X 0,Y 453.457,Z 149.497,A -85,B 0,C 180,E1 -8318.312,E2 -8318.312} C_VEL
LIN {X 0,Y 453.493,Z 149.492,A -85,B 0,C 180,E1 -8320.609,E2 -8320.609} C_VEL
LIN {X 0,Y 453.46,Z 149.496,A -85,B 0,C 180,E1 -8324.222,E2 -8324.222} C_VEL
LIN {X 0,Y 453.448,Z 149.5,A -85,B 0,C 180,E1 -8327.003,E2 -8327.003} C_VEL
LIN {X 0,Y 453.47,Z 149.501,A -85,B 0,C 180,E1 -8329.413,E2 -8329.413} C_VEL
LIN {X 0,Y 453.452,Z 149.5,A -85,B 0,C 180,E1 -8332.81,E2 -8332.81} C_VEL
LIN {X 0,Y 453.469,Z 149.495,A -85,B 0,C 180,E1 -8336.087,E2 -8336.087} C_VEL
LIN {X 0,Y 453.474,Z 149.502,A -85,B 0,C 180,E1 -8339.241,E2 -8339.241} C_VEL
LIN {X 0,Y 453.49,Z 149.494,A -85,B 0,C 180,E1 -8342.295,E2 -8342.295} C_VEL
LIN {X 0,Y 453.518,Z 149.613,A -85,B 0,C 180,E1 -8344.216,E2 -8344.216} C_VEL
LIN {X 0,Y 455.782,Z 161.293,A -85,B 0,C 180,E1 -8346.606,E2 -8346.606} C_VEL
LIN {X 0,Y 455.182,Z 175.044,A -85,B 0,C 180,E1 -8349.199,E2 -8349.199} C_VEL
LIN {X 0,Y 454.412,Z 192.26,A -85,B 0,C 180,E1 -8352.401,E2 -8352.401} C_VEL
LIN {X 0,Y 454.396,Z 192.489,A -85,B 0,C 180,E1 -8352.443,E2 -8352.443} C_VEL
LIN {X 0,Y 457.647,Z 213.522,A -85,B 0,C 180,E1 -8352.909,E2 -8352.909} C_VEL
LIN {X 0,Y 456.916,Z 300.591,A -85,B 0,C 180,E1 -8354.299,E2 -8354.299} C_VEL
LIN {X 0,Y 456.493,Z 313.846,A -85,B 0,C 180,E1 -8354.685,E2 -8354.685} C_VEL
LIN {X 0,Y 456.02,Z 325.999,A -85,B 0,C 180,E1 -8355.211,E2 -8355.211} C_VEL
LIN {X 0,Y 455.442,Z 338.261,A -85,B 0,C 180,E1 -8355.934,E2 -8355.934} C_VEL
LIN {X 0,Y 454.837,Z 349.217,A -85,B 0,C 180,E1 -8356.77,E2 -8356.77} C_VEL
LIN {X 0,Y 454.329,Z 360.289,A -85,B 0,C 180,E1 -8357.833,E2 -8357.833} C_VEL
LIN {X 0,Y 453.818,Z 368.821,A -85,B 0,C 180,E1 -8358.838,E2 -8358.838} C_VEL
LIN {X 0,Y 453.424,Z 376.695,A -85,B 0,C 180,E1 -8359.958,E2 -8359.958} C_VEL
LIN {X 0,Y 453.005,Z 384.383,A -85,B 0,C 180,E1 -8361.3,E2 -8361.3} C_VEL
LIN {X 0,Y 452.717,Z 391.472,A -85,B 0,C 180,E1 -8362.866,E2 -8362.866} C_VEL
LIN {X 0,Y 452.562,Z 396.189,A -85,B 0,C 180,E1 -8364.207,E2 -8364.207} C_VEL
LIN {X 0,Y 452.485,Z 399.792,A -85,B 0,C 180,E1 -8365.546,E2 -8365.546} C_VEL
LIN {X 0,Y 452.455,Z 401.651,A -85,B 0,C 180,E1 -8366.438,E2 -8366.438} C_VEL
LIN {X 0,Y 452.503,Z 403.046,A -85,B 0,C 180,E1 -8367.329,E2 -8367.329} C_VEL
LIN {X 0,Y 452.404,Z 404.645,A -85,B 0,C 180,E1 -8369.11,E2 -8369.11} C_VEL
LIN {X 0,Y 452.408,Z 404.861,A -85,B 0,C 180,E1 -8370,E2 -8370} C_VEL
LIN {X 0,Y 452.436,Z 404.038,A -85,B 0,C 180,E1 -8371.78,E2 -8371.78} C_VEL
LIN {X 0,Y 452.503,Z 403.046,A -85,B 0,C 180,E1 -8372.671,E2 -8372.671} C_VEL
LIN {X 0,Y 452.455,Z 401.65,A -85,B 0,C 180,E1 -8373.562,E2 -8373.562} C_VEL
LIN {X 0,Y 452.545,Z 398.718,A -85,B 0,C 180,E1 -8374.9,E2 -8374.9} C_VEL
LIN {X 0,Y 452.611,Z 394.211,A -85,B 0,C 180,E1 -8376.396,E2 -8376.396} C_VEL
LIN {X 0,Y 452.811,Z 388.642,A -85,B 0,C 180,E1 -8377.805,E2 -8377.805} C_VEL
LIN {X 0,Y 453.101,Z 381.971,A -85,B 0,C 180,E1 -8379.148,E2 -8379.148} C_VEL
LIN {X 0,Y 453.516,Z 373.694,A -85,B 0,C 180,E1 -8380.491,E2 -8380.491} C_VEL
LIN {X 0,Y 454.055,Z 365.211,A -85,B 0,C 180,E1 -8381.608,E2 -8381.608} C_VEL
LIN {X 0,Y 454.646,Z 355.56,A -85,B 0,C 180,E1 -8382.645,E2 -8382.645} C_VEL
LIN {X 0,Y 455.049,Z 345.783,A -85,B 0,C 180,E1 -8383.509,E2 -8383.509} C_VEL
LIN {X 0,Y 455.595,Z 334.752,A -85,B 0,C 180,E1 -8384.289,E2 -8384.289} C_VEL
LIN {X 0,Y 456.159,Z 322.526,A -85,B 0,C 180,E1 -8384.955,E2 -8384.955} C_VEL
LIN {X 0,Y 456.647,Z 310.608,A -85,B 0,C 180,E1 -8385.424,E2 -8385.424} C_VEL
LIN {X 0,Y 456.96,Z 297.576,A -85,B 0,C 180,E1 -8385.757,E2 -8385.757} C_VEL
LIN {X 0,Y 457.558,Z 211.978,A -85,B 0,C 180,E1 -8387.115,E2 -8387.115} C_VEL
LIN {X 0,Y 454.4,Z 192.457,A -85,B 0,C 180,E1 -8387.559,E2 -8387.559} C_VEL
LIN {X 0,Y 455.119,Z 176.267,A -85,B 0,C 180,E1 -8390.567,E2 -8390.567} C_VEL
LIN {X 0,Y 455.794,Z 162.517,A -85,B 0,C 180,E1 -8393.153,E2 -8393.153} C_VEL
LIN {X 0,Y 454.935,Z 156.829,A -85,B 0,C 180,E1 -8394.293,E2 -8394.293} C_VEL
LIN {X 0,Y 453.499,Z 149.496,A -85,B 0,C 180,E1 -8395.807,E2 -8395.807} C_VEL
LIN {X 0,Y 453.464,Z 149.496,A -85,B 0,C 180,E1 -8398.715,E2 -8398.715} C_VEL
LIN {X 0,Y 453.457,Z 149.496,A -85,B 0,C 180,E1 -8401.8,E2 -8401.8} C_VEL
LIN {X 0,Y 453.477,Z 149.5,A -85,B 0,C 180,E1 -8404.989,E2 -8404.989} C_VEL
LIN {X 0,Y 453.458,Z 149.498,A -85,B 0,C 180,E1 -8408.312,E2 -8408.312} C_VEL
LIN {X 0,Y 453.47,Z 149.501,A -85,B 0,C 180,E1 -8410.611,E2 -8410.611} C_VEL
LIN {X 0,Y 453.46,Z 149.499,A -85,B 0,C 180,E1 -8414.222,E2 -8414.222} C_VEL
LIN {X 0,Y 453.448,Z 149.499,A -85,B 0,C 180,E1 -8417.003,E2 -8417.003} C_VEL
LIN {X 0,Y 453.493,Z 149.492,A -85,B 0,C 180,E1 -8419.409,E2 -8419.409} C_VEL
LIN {X 0,Y 453.449,Z 149.499,A -85,B 0,C 180,E1 -8422.81,E2 -8422.81} C_VEL
LIN {X 0,Y 453.476,Z 149.499,A -85,B 0,C 180,E1 -8426.087,E2 -8426.087} C_VEL
LIN {X 0,Y 453.474,Z 149.494,A -85,B 0,C 180,E1 -8429.24,E2 -8429.24} C_VEL
LIN {X 0,Y 453.507,Z 149.495,A -85,B 0,C 180,E1 -8432.296,E2 -8432.296} C_VEL
LIN {X 0,Y 453.5,Z 149.492,A -85,B 0,C 180,E1 -8435.265,E2 -8435.265} C_VEL
LIN {X 0,Y 453.48,Z 149.495,A -85,B 0,C 180,E1 -8438.415,E2 -8438.415} C_VEL
LIN {X 0,Y 453.522,Z 149.488,A -85,B 0,C 180,E1 -8441.009,E2 -8441.009} C_VEL
LIN {X 0,Y 453.568,Z 149.488,A -85,B 0,C 180,E1 -8443.88,E2 -8443.88} C_VEL
LIN {X 0,Y 453.563,Z 149.489,A -85,B 0,C 180,E1 -8447.471,E2 -8447.471} C_VEL
LIN {X 0,Y 453.59,Z 149.482,A -85,B 0,C 180,E1 -8451.087,E2 -8451.087} C_VEL
LIN {X 0,Y 453.669,Z 149.473,A -85,B 0,C 180,E1 -8453.775,E2 -8453.775} C_VEL
LIN {X 0,Y 453.764,Z 149.466,A -85,B 0,C 180,E1 -8457.337,E2 -8457.337} C_VEL
LIN {X 0,Y 453.822,Z 149.451,A -85,B 0,C 180,E1 -8460,E2 -8460} C_VEL
LIN {X 0,Y 453.764,Z 149.46,A -85,B 0,C 180,E1 -8462.663,E2 -8462.663} C_VEL
LIN {X 0,Y 453.653,Z 149.472,A -85,B 0,C 180,E1 -8466.226,E2 -8466.226} C_VEL
LIN {X 0,Y 453.591,Z 149.487,A -85,B 0,C 180,E1 -8468.913,E2 -8468.913} C_VEL
LIN {X 0,Y 453.563,Z 149.487,A -85,B 0,C 180,E1 -8472.529,E2 -8472.529} C_VEL
LIN {X 0,Y 453.545,Z 149.487,A -85,B 0,C 180,E1 -8476.196,E2 -8476.196} C_VEL
LIN {X 0,Y 453.521,Z 149.491,A -85,B 0,C 180,E1 -8479.041,E2 -8479.041} C_VEL
LIN {X 0,Y 453.476,Z 149.494,A -85,B 0,C 180,E1 -8481.836,E2 -8481.836} C_VEL
LIN {X 0,Y 453.513,Z 149.494,A -85,B 0,C 180,E1 -8484.735,E2 -8484.735} C_VEL
LIN {X 0,Y 453.532,Z 149.489,A -85,B 0,C 180,E1 -8487.96,E2 -8487.96} C_VEL
LIN {X 0,Y 453.466,Z 149.495,A -85,B 0,C 180,E1 -8491.525,E2 -8491.525} C_VEL
LIN {X 0,Y 453.488,Z 149.494,A -85,B 0,C 180,E1 -8494.778,E2 -8494.778} C_VEL
LIN {X 0,Y 453.465,Z 149.5,A -85,B 0,C 180,E1 -8498.312,E2 -8498.312} C_VEL
LIN {X 0,Y 453.495,Z 149.493,A -85,B 0,C 180,E1 -8500.609,E2 -8500.609} C_VEL
LIN {X 0,Y 453.456,Z 149.497,A -85,B 0,C 180,E1 -8503.244,E2 -8503.244} C_VEL
LIN {X 0,Y 453.467,Z 149.502,A -85,B 0,C 180,E1 -8505.779,E2 -8505.779} C_VEL
LIN {X 0,Y 453.48,Z 149.496,A -85,B 0,C 180,E1 -8508.21,E2 -8508.21} C_VEL
LIN {X 0,Y 453.488,Z 149.492,A -85,B 0,C 180,E1 -8510.795,E2 -8510.795} C_VEL
LIN {X 0,Y 453.455,Z 149.5,A -85,B 0,C 180,E1 -8513.917,E2 -8513.917} C_VEL
LIN {X 0,Y 453.48,Z 149.496,A -85,B 0,C 180,E1 -8517.151,E2 -8517.151} C_VEL
LIN {X 0,Y 453.476,Z 149.494,A -85,B 0,C 180,E1 -8520.268,E2 -8520.268} C_VEL
LIN {X 0,Y 453.509,Z 149.497,A -85,B 0,C 180,E1 -8523.294,E2 -8523.294} C_VEL
LIN {X 0,Y 453.505,Z 149.493,A -85,B 0,C 180,E1 -8526.239,E2 -8526.239} C_VEL
LIN {X 0,Y 453.544,Z 149.632,A -85,B 0,C 180,E1 -8527.538,E2 -8527.538} C_VEL
LIN {X 0,Y 455.051,Z 158.151,A -85,B 0,C 180,E1 -8529.429,E2 -8529.429} C_VEL
LIN {X 0,Y 454.667,Z 170.597,A -85,B 0,C 180,E1 -8531.992,E2 -8531.992} C_VEL
LIN {X 0,Y 454.533,Z 173.077,A -85,B 0,C 180,E1 -8532.491,E2 -8532.491} C_VEL
LIN {X 0,Y 457.768,Z 189.819,A -85,B 0,C 180,E1 -8532.903,E2 -8532.903} C_VEL
LIN {X 0,Y 457.464,Z 235.815,A -85,B 0,C 180,E1 -8533.63,E2 -8533.63} C_VEL
LIN {X 0,Y 456.896,Z 241.657,A -85,B 0,C 180,E1 -8533.703,E2 -8533.703} C_VEL
LIN {X 0,Y 454.051,Z 251.15,A -85,B 0,C 180,E1 -8533.75,E2 -8533.75} C_VEL
LIN {X 0,Y 451.111,Z 260.644,A -85,B 0,C 180,E1 -8533.794,E2 -8533.794} C_VEL
LIN {X 0,Y 450.4,Z 266.495,A -85,B 0,C 180,E1 -8533.863,E2 -8533.863} C_VEL
LIN {X 0,Y 450.156,Z 283.282,A -85,B 0,C 180,E1 -8534.173,E2 -8534.173} C_VEL
LIN {X 0,Y 449.735,Z 296.389,A -85,B 0,C 180,E1 -8534.594,E2 -8534.594} C_VEL
LIN {X 0,Y 449.307,Z 308.292,A -85,B 0,C 180,E1 -8535.159,E2 -8535.159} C_VEL
LIN {X 0,Y 448.778,Z 320.729,A -85,B 0,C 180,E1 -8535.952,E2 -8535.952} C_VEL
LIN {X 0,Y 448.293,Z 330.453,A -85,B 0,C 180,E1 -8536.74,E2 -8536.74} C_VEL
LIN {X 0,Y 447.722,Z 340.762,A -85,B 0,C 180,E1 -8537.766,E2 -8537.766} C_VEL
LIN {X 0,Y 447.132,Z 349.957,A -85,B 0,C 180,E1 -8538.899,E2 -8538.899} C_VEL
LIN {X 0,Y 446.565,Z 358.883,A -85,B 0,C 180,E1 -8540.26,E2 -8540.26} C_VEL
LIN {X 0,Y 446.133,Z 366.068,A -85,B 0,C 180,E1 -8541.621,E2 -8541.621} C_VEL
LIN {X 0,Y 445.847,Z 372.02,A -85,B 0,C 180,E1 -8543.042,E2 -8543.042} C_VEL
LIN {X 0,Y 445.65,Z 376.941,A -85,B 0,C 180,E1 -8544.57,E2 -8544.57} C_VEL
LIN {X 0,Y 445.491,Z 379.233,A -85,B 0,C 180,E1 -8545.476,E2 -8545.476} C_VEL
LIN {X 0,Y 445.516,Z 381.095,A -85,B 0,C 180,E1 -8546.382,E2 -8546.382} C_VEL
LIN {X 0,Y 445.471,Z 382.5,A -85,B 0,C 180,E1 -8547.287,E2 -8547.287} C_VEL
LIN {X 0,Y 445.343,Z 384.116,A -85,B 0,C 180,E1 -8549.096,E2 -8549.096} C_VEL
LIN {X 0,Y 445.319,Z 384.352,A -85,B 0,C 180,E1 -8550,E2 -8550} C_VEL
LIN {X 0,Y 445.342,Z 384.165,A -85,B 0,C 180,E1 -8550.904,E2 -8550.904} C_VEL
LIN {X 0,Y 445.471,Z 382.612,A -85,B 0,C 180,E1 -8552.713,E2 -8552.713} C_VEL
LIN {X 0,Y 445.513,Z 381.256,A -85,B 0,C 180,E1 -8553.618,E2 -8553.618} C_VEL
LIN {X 0,Y 445.536,Z 378.391,A -85,B 0,C 180,E1 -8554.977,E2 -8554.977} C_VEL
LIN {X 0,Y 445.779,Z 374.501,A -85,B 0,C 180,E1 -8556.336,E2 -8556.336} C_VEL
LIN {X 0,Y 445.961,Z 369.486,A -85,B 0,C 180,E1 -8557.698,E2 -8557.698} C_VEL
LIN {X 0,Y 446.311,Z 363.173,A -85,B 0,C 180,E1 -8559.06,E2 -8559.06} C_VEL
LIN {X 0,Y 446.774,Z 355.269,A -85,B 0,C 180,E1 -8560.422,E2 -8560.422} C_VEL
LIN {X 0,Y 447.266,Z 347.211,A -85,B 0,C 180,E1 -8561.557,E2 -8561.557} C_VEL
LIN {X 0,Y 447.923,Z 337.375,A -85,B 0,C 180,E1 -8562.689,E2 -8562.689} C_VEL
LIN {X 0,Y 448.495,Z 326.466,A -85,B 0,C 180,E1 -8563.698,E2 -8563.698} C_VEL
LIN {X 0,Y 449.012,Z 315.482,A -85,B 0,C 180,E1 -8564.503,E2 -8564.503} C_VEL
LIN {X 0,Y 449.549,Z 303.51,A -85,B 0,C 180,E1 -8565.18,E2 -8565.18} C_VEL
LIN {X 0,Y 450.001,Z 290.381,A -85,B 0,C 180,E1 -8565.716,E2 -8565.716} C_VEL
LIN {X 0,Y 450.287,Z 277.177,A -85,B 0,C 180,E1 -8566.054,E2 -8566.054} C_VEL
LIN {X 0,Y 451.006,Z 190.728,A -85,B 0,C 180,E1 -8567.445,E2 -8567.445} C_VEL
LIN {X 0,Y 447.653,Z 173.271,A -85,B 0,C 180,E1 -8567.874,E2 -8567.874} C_VEL
LIN {X 0,Y 448.168,Z 159.853,A -85,B 0,C 180,E1 -8570.661,E2 -8570.661} C_VEL
LIN {X 0,Y 446.487,Z 150.37,A -85,B 0,C 180,E1 -8572.806,E2 -8572.806} C_VEL
LIN {X 0,Y 446.477,Z 150.369,A -85,B 0,C 180,E1 -8576.202,E2 -8576.202} C_VEL
LIN {X 0,Y 446.45,Z 150.371,A -85,B 0,C 180,E1 -8579.209,E2 -8579.209} C_VEL
LIN {X 0,Y 446.421,Z 150.378,A -85,B 0,C 180,E1 -8582.361,E2 -8582.361} C_VEL
LIN {X 0,Y 446.419,Z 150.373,A -85,B 0,C 180,E1 -8585.626,E2 -8585.626} C_VEL
LIN {X 0,Y 446.439,Z 150.371,A -85,B 0,C 180,E1 -8589.027,E2 -8589.027} C_VEL
LIN {X 0,Y 446.435,Z 150.379,A -85,B 0,C 180,E1 -8592.277,E2 -8592.277} C_VEL
LIN {X 0,Y 446.454,Z 150.369,A -85,B 0,C 180,E1 -8595.103,E2 -8595.103} C_VEL
LIN {X 0,Y 446.429,Z 150.373,A -85,B 0,C 180,E1 -8598.609,E2 -8598.609} C_VEL
LIN {X 0,Y 446.444,Z 150.37,A -85,B 0,C 180,E1 -8600.973,E2 -8600.973} C_VEL
LIN {X 0,Y 446.419,Z 150.375,A -85,B 0,C 180,E1 -8604.374,E2 -8604.374} C_VEL
LIN {X 0,Y 446.422,Z 150.378,A -85,B 0,C 180,E1 -8607.638,E2 -8607.638} C_VEL
LIN {X 0,Y 446.448,Z 150.369,A -85,B 0,C 180,E1 -8610.79,E2 -8610.79} C_VEL
LIN {X 0,Y 446.477,Z 150.37,A -85,B 0,C 180,E1 -8613.848,E2 -8613.848} C_VEL
LIN {X 0,Y 446.428,Z 150.372,A -85,B 0,C 180,E1 -8616.823,E2 -8616.823} C_VEL
LIN {X 0,Y 446.444,Z 150.374,A -85,B 0,C 180,E1 -8619.737,E2 -8619.737} C_VEL
LIN {X 0,Y 446.463,Z 150.368,A -85,B 0,C 180,E1 -8622.597,E2 -8622.597} C_VEL
LIN {X 0,Y 446.47,Z 150.372,A -85,B 0,C 180,E1 -8625.412,E2 -8625.412} C_VEL
LIN {X 0,Y 446.517,Z 150.361,A -85,B 0,C 180,E1 -8628.193,E2 -8628.193} C_VEL
LIN {X 0,Y 446.6,Z 150.351,A -85,B 0,C 180,E1 -8631.858,E2 -8631.858} C_VEL
LIN {X 0,Y 446.641,Z 150.348,A -85,B 0,C 180,E1 -8634.582,E2 -8634.582} C_VEL
LIN {X 0,Y 446.708,Z 150.34,A -85,B 0,C 180,E1 -8637.295,E2 -8637.295} C_VEL
LIN {X 0,Y 446.792,Z 150.327,A -85,B 0,C 180,E1 -8640,E2 -8640} C_VEL
LIN {X 0,Y 446.707,Z 150.345,A -85,B 0,C 180,E1 -8642.705,E2 -8642.705} C_VEL
LIN {X 0,Y 446.638,Z 150.349,A -85,B 0,C 180,E1 -8646.324,E2 -8646.324} C_VEL
LIN {X 0,Y 446.536,Z 150.36,A -85,B 0,C 180,E1 -8649.055,E2 -8649.055} C_VEL
LIN {X 0,Y 446.52,Z 150.364,A -85,B 0,C 180,E1 -8652.73,E2 -8652.73} C_VEL
LIN {X 0,Y 446.495,Z 150.37,A -85,B 0,C 180,E1 -8656.228,E2 -8656.228} C_VEL
LIN {X 0,Y 446.467,Z 150.367,A -85,B 0,C 180,E1 -8659.303,E2 -8659.303} C_VEL
LIN {X 0,Y 446.417,Z 150.38,A -85,B 0,C 180,E1 -8662.2,E2 -8662.2} C_VEL
LIN {X 0,Y 446.443,Z 150.37,A -85,B 0,C 180,E1 -8665.153,E2 -8665.153} C_VEL
LIN {X 0,Y 446.484,Z 150.37,A -85,B 0,C 180,E1 -8668.179,E2 -8668.179} C_VEL
LIN {X 0,Y 446.418,Z 150.38,A -85,B 0,C 180,E1 -8671.775,E2 -8671.775} C_VEL
LIN {X 0,Y 446.427,Z 150.372,A -85,B 0,C 180,E1 -8674.523,E2 -8674.523} C_VEL
LIN {X 0,Y 446.41,Z 150.377,A -85,B 0,C 180,E1 -8678.079,E2 -8678.079} C_VEL
LIN {X 0,Y 446.422,Z 150.374,A -85,B 0,C 180,E1 -8680.917,E2 -8680.917} C_VEL
LIN {X 0,Y 446.398,Z 150.379,A -85,B 0,C 180,E1 -8683.847,E2 -8683.847} C_VEL
LIN {X 0,Y 446.397,Z 150.376,A -85,B 0,C 180,E1 -8686.404,E2 -8686.404} C_VEL
LIN {X 0,Y 446.404,Z 150.379,A -85,B 0,C 180,E1 -8689.086,E2 -8689.086} C_VEL
LIN {X 0,Y 446.406,Z 150.375,A -85,B 0,C 180,E1 -8692.121,E2 -8692.121} C_VEL
LIN {X 0,Y 446.423,Z 150.376,A -85,B 0,C 180,E1 -8695.477,E2 -8695.477} C_VEL
LIN {X 0,Y 446.415,Z 150.377,A -85,B 0,C 180,E1 -8698.7,E2 -8698.7} C_VEL
LIN {X 0,Y 446.447,Z 150.37,A -85,B 0,C 180,E1 -8701.831,E2 -8701.831} C_VEL
LIN {X 0,Y 446.449,Z 150.421,A -85,B 0,C 180,E1 -8703.972,E2 -8703.972} C_VEL
LIN {X 0,Y 448.78,Z 162.382,A -85,B 0,C 180,E1 -8706.463,E2 -8706.463} C_VEL
LIN {X 0,Y 448.686,Z 167.939,A -85,B 0,C 180,E1 -8707.541,E2 -8707.541} C_VEL
LIN {X 0,Y 447.762,Z 186.115,A -85,B 0,C 180,E1 -8710.993,E2 -8710.993} C_VEL
LIN {X 0,Y 447.464,Z 192.351,A -85,B 0,C 180,E1 -8712.162,E2 -8712.162} C_VEL
LIN {X 0,Y 450.84,Z 213.377,A -85,B 0,C 180,E1 -8712.643,E2 -8712.643} C_VEL
LIN {X 0,Y 450.091,Z 300.44,A -85,B 0,C 180,E1 -8714.055,E2 -8714.055} C_VEL
LIN {X 0,Y 449.698,Z 312.929,A -85,B 0,C 180,E1 -8714.418,E2 -8714.418} C_VEL
LIN {X 0,Y 449.168,Z 325.842,A -85,B 0,C 180,E1 -8714.981,E2 -8714.981} C_VEL
LIN {X 0,Y 448.546,Z 338.102,A -85,B 0,C 180,E1 -8715.713,E2 -8715.713} C_VEL
LIN {X 0,Y 447.845,Z 350.032,A -85,B 0,C 180,E1 -8716.647,E2 -8716.647} C_VEL
LIN {X 0,Y 447.311,Z 361.172,A -85,B 0,C 180,E1 -8717.754,E2 -8717.754} C_VEL
LIN {X 0,Y 446.704,Z 370.337,A -85,B 0,C 180,E1 -8718.888,E2 -8718.888} C_VEL
LIN {X 0,Y 446.211,Z 379.269,A -85,B 0,C 180,E1 -8720.252,E2 -8720.252} C_VEL
LIN {X 0,Y 445.842,Z 386.458,A -85,B 0,C 180,E1 -8721.616,E2 -8721.616} C_VEL
LIN {X 0,Y 445.634,Z 391.31,A -85,B 0,C 180,E1 -8722.752,E2 -8722.752} C_VEL
LIN {X 0,Y 445.485,Z 395.468,A -85,B 0,C 180,E1 -8723.937,E2 -8723.937} C_VEL
LIN {X 0,Y 445.411,Z 399.631,A -85,B 0,C 180,E1 -8725.475,E2 -8725.475} C_VEL
LIN {X 0,Y 445.354,Z 401.489,A -85,B 0,C 180,E1 -8726.381,E2 -8726.381} C_VEL
LIN {X 0,Y 445.427,Z 402.884,A -85,B 0,C 180,E1 -8727.287,E2 -8727.287} C_VEL
LIN {X 0,Y 445.316,Z 404.484,A -85,B 0,C 180,E1 -8729.096,E2 -8729.096} C_VEL
LIN {X 0,Y 445.317,Z 404.699,A -85,B 0,C 180,E1 -8730,E2 -8730} C_VEL
LIN {X 0,Y 445.355,Z 403.876,A -85,B 0,C 180,E1 -8731.809,E2 -8731.809} C_VEL
LIN {X 0,Y 445.427,Z 402.883,A -85,B 0,C 180,E1 -8732.713,E2 -8732.713} C_VEL
LIN {X 0,Y 445.354,Z 401.487,A -85,B 0,C 180,E1 -8733.619,E2 -8733.619} C_VEL
LIN {X 0,Y 445.473,Z 398.555,A -85,B 0,C 180,E1 -8734.978,E2 -8734.978} C_VEL
LIN {X 0,Y 445.574,Z 393.154,A -85,B 0,C 180,E1 -8736.748,E2 -8736.748} C_VEL
LIN {X 0,Y 445.786,Z 387.467,A -85,B 0,C 180,E1 -8738.157,E2 -8738.157} C_VEL
LIN {X 0,Y 446.135,Z 380.571,A -85,B 0,C 180,E1 -8739.521,E2 -8739.521} C_VEL
LIN {X 0,Y 446.585,Z 371.942,A -85,B 0,C 180,E1 -8740.885,E2 -8740.885} C_VEL
LIN {X 0,Y 447.188,Z 363.096,A -85,B 0,C 180,E1 -8742.019,E2 -8742.019} C_VEL
LIN {X 0,Y 447.7,Z 354.288,A -85,B 0,C 180,E1 -8742.953,E2 -8742.953} C_VEL
LIN {X 0,Y 448.283,Z 342.759,A -85,B 0,C 180,E1 -8743.948,E2 -8743.948} C_VEL
LIN {X 0,Y 448.893,Z 330.89,A -85,B 0,C 180,E1 -8744.739,E2 -8744.739} C_VEL
LIN {X 0,Y 449.415,Z 318.538,A -85,B 0,C 180,E1 -8745.359,E2 -8745.359} C_VEL
LIN {X 0,Y 449.955,Z 305.859,A -85,B 0,C 180,E1 -8745.805,E2 -8745.805} C_VEL
LIN {X 0,Y 450.206,Z 292.582,A -85,B 0,C 180,E1 -8746.087,E2 -8746.087} C_VEL
LIN {X 0,Y 450.719,Z 212.404,A -85,B 0,C 180,E1 -8747.373,E2 -8747.373} C_VEL
LIN {X 0,Y 447.447,Z 192.208,A -85,B 0,C 180,E1 -8747.856,E2 -8747.856} C_VEL
LIN {X 0,Y 448.296,Z 174.854,A -85,B 0,C 180,E1 -8751.135,E2 -8751.135} C_VEL
LIN {X 0,Y 448.85,Z 163.604,A -85,B 0,C 180,E1 -8753.288,E2 -8753.288} C_VEL
LIN {X 0,Y 447.331,Z 154.795,A -85,B 0,C 180,E1 -8755.1,E2 -8755.1} C_VEL
LIN {X 0,Y 446.444,Z 150.374,A -85,B 0,C 180,E1 -8756.063,E2 -8756.063} C_VEL
LIN {X 0,Y 446.422,Z 150.377,A -85,B 0,C 180,E1 -8759.211,E2 -8759.211} C_VEL
LIN {X 0,Y 446.415,Z 150.375,A -85,B 0,C 180,E1 -8762.362,E2 -8762.362} C_VEL
LIN {X 0,Y 446.418,Z 150.373,A -85,B 0,C 180,E1 -8765.626,E2 -8765.626} C_VEL
LIN {X 0,Y 446.422,Z 150.377,A -85,B 0,C 180,E1 -8769.029,E2 -8769.029} C_VEL
LIN {X 0,Y 446.419,Z 150.376,A -85,B 0,C 180,E1 -8772.275,E2 -8772.275} C_VEL
LIN {X 0,Y 446.45,Z 150.371,A -85,B 0,C 180,E1 -8775.104,E2 -8775.104} C_VEL
LIN {X 0,Y 446.418,Z 150.379,A -85,B 0,C 180,E1 -8778.608,E2 -8778.608} C_VEL
LIN {X 0,Y 446.424,Z 150.374,A -85,B 0,C 180,E1 -8780.971,E2 -8780.971} C_VEL
LIN {X 0,Y 446.417,Z 150.38,A -85,B 0,C 180,E1 -8784.374,E2 -8784.374} C_VEL
LIN {X 0,Y 446.422,Z 150.374,A -85,B 0,C 180,E1 -8787.638,E2 -8787.638} C_VEL
LIN {X 0,Y 446.436,Z 150.371,A -85,B 0,C 180,E1 -8790.79,E2 -8790.79} C_VEL
LIN {X 0,Y 446.439,Z 150.376,A -85,B 0,C 180,E1 -8793.846,E2 -8793.846} C_VEL
LIN {X 0,Y 446.425,Z 150.372,A -85,B 0,C 180,E1 -8796.823,E2 -8796.823} C_VEL
LIN {X 0,Y 446.443,Z 150.376,A -85,B 0,C 180,E1 -8799.737,E2 -8799.737} C_VEL
LIN {X 0,Y 446.456,Z 150.368,A -85,B 0,C 180,E1 -8802.597,E2 -8802.597} C_VEL
LIN {X 0,Y 446.47,Z 150.371,A -85,B 0,C 180,E1 -8805.412,E2 -8805.412} C_VEL
LIN {X 0,Y 446.517,Z 150.362,A -85,B 0,C 180,E1 -8808.193,E2 -8808.193} C_VEL
LIN {X 0,Y 446.6,Z 150.353,A -85,B 0,C 180,E1 -8811.858,E2 -8811.858} C_VEL
LIN {X 0,Y 446.642,Z 150.345,A -85,B 0,C 180,E1 -8814.583,E2 -8814.583} C_VEL
LIN {X 0,Y 446.707,Z 150.345,A -85,B 0,C 180,E1 -8817.295,E2 -8817.295} C_VEL
LIN {X 0,Y 446.792,Z 150.327,A -85,B 0,C 180,E1 -8820,E2 -8820} C_VEL
LIN {X 0,Y 446.708,Z 150.339,A -85,B 0,C 180,E1 -8822.705,E2 -8822.705} C_VEL
LIN {X 0,Y 446.621,Z 150.348,A -85,B 0,C 180,E1 -8826.324,E2 -8826.324} C_VEL
LIN {X 0,Y 446.536,Z 150.365,A -85,B 0,C 180,E1 -8829.055,E2 -8829.055} C_VEL
LIN {X 0,Y 446.521,Z 150.366,A -85,B 0,C 180,E1 -8832.73,E2 -8832.73} C_VEL
LIN {X 0,Y 446.496,Z 150.365,A -85,B 0,C 180,E1 -8836.228,E2 -8836.228} C_VEL
LIN {X 0,Y 446.47,Z 150.368,A -85,B 0,C 180,E1 -8839.303,E2 -8839.303} C_VEL
LIN {X 0,Y 446.418,Z 150.376,A -85,B 0,C 180,E1 -8842.2,E2 -8842.2} C_VEL
LIN {X 0,Y 446.457,Z 150.369,A -85,B 0,C 180,E1 -8845.152,E2 -8845.152} C_VEL
LIN {X 0,Y 446.485,Z 150.37,A -85,B 0,C 180,E1 -8848.179,E2 -8848.179} C_VEL
LIN {X 0,Y 446.419,Z 150.375,A -85,B 0,C 180,E1 -8851.775,E2 -8851.775} C_VEL
LIN {X 0,Y 446.43,Z 150.375,A -85,B 0,C 180,E1 -8854.523,E2 -8854.523} C_VEL
LIN {X 0,Y 446.416,Z 150.381,A -85,B 0,C 180,E1 -8858.08,E2 -8858.08} C_VEL
LIN {X 0,Y 446.427,Z 150.372,A -85,B 0,C 180,E1 -8860.918,E2 -8860.918} C_VEL
LIN {X 0,Y 446.418,Z 150.38,A -85,B 0,C 180,E1 -8863.844,E2 -8863.844} C_VEL
LIN {X 0,Y 446.401,Z 150.377,A -85,B 0,C 180,E1 -8866.404,E2 -8866.404} C_VEL
LIN {X 0,Y 446.428,Z 150.373,A -85,B 0,C 180,E1 -8869.083,E2 -8869.083} C_VEL
LIN {X 0,Y 446.409,Z 150.377,A -85,B 0,C 180,E1 -8872.121,E2 -8872.121} C_VEL
LIN {X 0,Y 446.425,Z 150.379,A -85,B 0,C 180,E1 -8875.477,E2 -8875.477} C_VEL
LIN {X 0,Y 446.417,Z 150.373,A -85,B 0,C 180,E1 -8878.7,E2 -8878.7} C_VEL
LIN {X 0,Y 446.487,Z 150.37,A -85,B 0,C 180,E1 -8881.822,E2 -8881.822} C_VEL
LIN {X 0,Y 446.46,Z 150.372,A -85,B 0,C 180,E1 -8884.848,E2 -8884.848} C_VEL
LIN {X 0,Y 446.492,Z 150.436,A -85,B 0,C 180,E1 -8887.316,E2 -8887.316} C_VEL
LIN {X 0,Y 448.104,Z 159.401,A -85,B 0,C 180,E1 -8889.336,E2 -8889.336} C_VEL
LIN {X 0,Y 447.697,Z 171.777,A -85,B 0,C 180,E1 -8891.915,E2 -8891.915} C_VEL
LIN {X 0,Y 447.622,Z 173.232,A -85,B 0,C 180,E1 -8892.212,E2 -8892.212} C_VEL
LIN {X 0,Y 451.052,Z 191.292,A -85,B 0,C 180,E1 -8892.661,E2 -8892.661} C_VEL
LIN {X 0,Y 450.4,Z 266.495,A -85,B 0,C 180,E1 -8893.863,E2 -8893.863} C_VEL
LIN {X 0,Y 449.667,Z 272.357,A -85,B 0,C 180,E1 -8893.93,E2 -8893.93} C_VEL
LIN {X 0,Y 446.652,Z 281.839,A -85,B 0,C 180,E1 -8894.006,E2 -8894.006} C_VEL
LIN {X 0,Y 443.641,Z 291.189,A -85,B 0,C 180,E1 -8894.166,E2 -8894.166} C_VEL
LIN {X 0,Y 442.896,Z 296.829,A -85,B 0,C 180,E1 -8894.362,E2 -8894.362} C_VEL
LIN {X 0,Y 442.464,Z 308.461,A -85,B 0,C 180,E1 -8894.924,E2 -8894.924} C_VEL
LIN {X 0,Y 441.903,Z 320.897,A -85,B 0,C 180,E1 -8895.729,E2 -8895.729} C_VEL
LIN {X 0,Y 441.349,Z 331.033,A -85,B 0,C 180,E1 -8896.565,E2 -8896.565} C_VEL
LIN {X 0,Y 440.798,Z 340.928,A -85,B 0,C 180,E1 -8897.57,E2 -8897.57} C_VEL
LIN {X 0,Y 440.158,Z 350.122,A -85,B 0,C 180,E1 -8898.72,E2 -8898.72} C_VEL
LIN {X 0,Y 439.563,Z 359.047,A -85,B 0,C 180,E1 -8900.103,E2 -8900.103} C_VEL
LIN {X 0,Y 439.104,Z 366.233,A -85,B 0,C 180,E1 -8901.486,E2 -8901.486} C_VEL
LIN {X 0,Y 438.827,Z 371.08,A -85,B 0,C 180,E1 -8902.639,E2 -8902.639} C_VEL
LIN {X 0,Y 438.664,Z 375.788,A -85,B 0,C 180,E1 -8904.022,E2 -8904.022} C_VEL
LIN {X 0,Y 438.416,Z 379.396,A -85,B 0,C 180,E1 -8905.403,E2 -8905.403} C_VEL
LIN {X 0,Y 438.418,Z 381.258,A -85,B 0,C 180,E1 -8906.324,E2 -8906.324} C_VEL
LIN {X 0,Y 438.4,Z 382.662,A -85,B 0,C 180,E1 -8907.243,E2 -8907.243} C_VEL
LIN {X 0,Y 438.256,Z 384.278,A -85,B 0,C 180,E1 -8909.081,E2 -8909.081} C_VEL
LIN {X 0,Y 438.231,Z 384.514,A -85,B 0,C 180,E1 -8910,E2 -8910} C_VEL
LIN {X 0,Y 438.256,Z 384.327,A -85,B 0,C 180,E1 -8910.919,E2 -8910.919} C_VEL
LIN {X 0,Y 438.4,Z 382.773,A -85,B 0,C 180,E1 -8912.757,E2 -8912.757} C_VEL
LIN {X 0,Y 438.413,Z 381.418,A -85,B 0,C 180,E1 -8913.676,E2 -8913.676} C_VEL
LIN {X 0,Y 438.479,Z 378.552,A -85,B 0,C 180,E1 -8915.057,E2 -8915.057} C_VEL
LIN {X 0,Y 438.705,Z 373.915,A -85,B 0,C 180,E1 -8916.668,E2 -8916.668} C_VEL
LIN {X 0,Y 439.016,Z 367.674,A -85,B 0,C 180,E1 -8918.284,E2 -8918.284} C_VEL
LIN {X 0,Y 439.454,Z 360.883,A -85,B 0,C 180,E1 -8919.667,E2 -8919.667} C_VEL
LIN {X 0,Y 439.965,Z 352.403,A -85,B 0,C 180,E1 -8921.051,E2 -8921.051} C_VEL
LIN {X 0,Y 440.602,Z 343.678,A -85,B 0,C 180,E1 -8922.201,E2 -8922.201} C_VEL
LIN {X 0,Y 441.226,Z 333.812,A -85,B 0,C 180,E1 -8923.266,E2 -8923.266} C_VEL
LIN {X 0,Y 441.739,Z 323.639,A -85,B 0,C 180,E1 -8924.158,E2 -8924.158} C_VEL
LIN {X 0,Y 442.333,Z 312.05,A -85,B 0,C 180,E1 -8924.962,E2 -8924.962} C_VEL
LIN {X 0,Y 442.859,Z 299.999,A -85,B 0,C 180,E1 -8925.592,E2 -8925.592} C_VEL
LIN {X 0,Y 443.246,Z 286.871,A -85,B 0,C 180,E1 -8926.08,E2 -8926.08} C_VEL
LIN {X 0,Y 443.529,Z 274.201,A -85,B 0,C 180,E1 -8926.365,E2 -8926.365} C_VEL
LIN {X 0,Y 444.204,Z 191.522,A -85,B 0,C 180,E1 -8927.71,E2 -8927.71} C_VEL
LIN {X 0,Y 440.704,Z 173.425,A -85,B 0,C 180,E1 -8928.166,E2 -8928.166} C_VEL
LIN {X 0,Y 441.218,Z 161.111,A -85,B 0,C 180,E1 -8930.757,E2 -8930.757} C_VEL
LIN {X 0,Y 439.427,Z 151.249,A -85,B 0,C 180,E1 -8933.038,E2 -8933.038} C_VEL
LIN {X 0,Y 439.431,Z 151.25,A -85,B 0,C 180,E1 -8936.603,E2 -8936.603} C_VEL
LIN {X 0,Y 439.383,Z 151.249,A -85,B 0,C 180,E1 -8939.726,E2 -8939.726} C_VEL
LIN {X 0,Y 439.373,Z 151.254,A -85,B 0,C 180,E1 -8942.946,E2 -8942.946} C_VEL
LIN {X 0,Y 439.374,Z 151.256,A -85,B 0,C 180,E1 -8946.287,E2 -8946.287} C_VEL
LIN {X 0,Y 439.402,Z 151.249,A -85,B 0,C 180,E1 -8949.849,E2 -8949.849} C_VEL
LIN {X 0,Y 439.383,Z 151.253,A -85,B 0,C 180,E1 -8952.627,E2 -8952.627} C_VEL
LIN {X 0,Y 439.404,Z 151.247,A -85,B 0,C 180,E1 -8955.271,E2 -8955.271} C_VEL
LIN {X 0,Y 439.389,Z 151.25,A -85,B 0,C 180,E1 -8958.743,E2 -8958.743} C_VEL
LIN {X 0,Y 439.374,Z 151.253,A -85,B 0,C 180,E1 -8961.607,E2 -8961.607} C_VEL
LIN {X 0,Y 439.399,Z 151.247,A -85,B 0,C 180,E1 -8964.844,E2 -8964.844} C_VEL
LIN {X 0,Y 439.372,Z 151.254,A -85,B 0,C 180,E1 -8968.139,E2 -8968.139} C_VEL
LIN {X 0,Y 439.432,Z 151.25,A -85,B 0,C 180,E1 -8971.598,E2 -8971.598} C_VEL
LIN {X 0,Y 439.404,Z 151.247,A -85,B 0,C 180,E1 -8974.415,E2 -8974.415} C_VEL
LIN {X 0,Y 439.364,Z 151.258,A -85,B 0,C 180,E1 -8977.424,E2 -8977.424} C_VEL
LIN {X 0,Y 439.441,Z 151.243,A -85,B 0,C 180,E1 -8980.663,E2 -8980.663} C_VEL
LIN {X 0,Y 439.462,Z 151.24,A -85,B 0,C 180,E1 -8984.224,E2 -8984.224} C_VEL
LIN {X 0,Y 439.483,Z 151.237,A -85,B 0,C 180,E1 -8988.001,E2 -8988.001} C_VEL
LIN {X 0,Y 439.547,Z 151.23,A -85,B 0,C 180,E1 -8991.726,E2 -8991.726} C_VEL
LIN {X 0,Y 439.616,Z 151.222,A -85,B 0,C 180,E1 -8994.496,E2 -8994.496} C_VEL
LIN {X 0,Y 439.636,Z 151.219,A -85,B 0,C 180,E1 -8998.168,E2 -8998.168} C_VEL
LIN {X 0,Y 439.762,Z 151.202,A -85,B 0,C 180,E1 -9000,E2 -9000} C_VEL
LIN {X 0,Y 439.654,Z 151.223,A -85,B 0,C 180,E1 -9002.749,E2 -9002.749} C_VEL
LIN {X 0,Y 439.61,Z 151.226,A -85,B 0,C 180,E1 -9006.425,E2 -9006.425} C_VEL
LIN {X 0,Y 439.498,Z 151.236,A -85,B 0,C 180,E1 -9009.202,E2 -9009.202} C_VEL
LIN {X 0,Y 439.465,Z 151.241,A -85,B 0,C 180,E1 -9012.938,E2 -9012.938} C_VEL
LIN {X 0,Y 439.445,Z 151.249,A -85,B 0,C 180,E1 -9016.348,E2 -9016.348} C_VEL
LIN {X 0,Y 439.401,Z 151.248,A -85,B 0,C 180,E1 -9019.626,E2 -9019.626} C_VEL
LIN {X 0,Y 439.363,Z 151.254,A -85,B 0,C 180,E1 -9022.576,E2 -9022.576} C_VEL
LIN {X 0,Y 439.396,Z 151.25,A -85,B 0,C 180,E1 -9025.585,E2 -9025.585} C_VEL
LIN {X 0,Y 439.416,Z 151.246,A -85,B 0,C 180,E1 -9028.674,E2 -9028.674} C_VEL
LIN {X 0,Y 439.369,Z 151.256,A -85,B 0,C 180,E1 -9032.031,E2 -9032.031} C_VEL
LIN {X 0,Y 439.392,Z 151.251,A -85,B 0,C 180,E1 -9035.34,E2 -9035.34} C_VEL
LIN {X 0,Y 439.368,Z 151.251,A -85,B 0,C 180,E1 -9038.597,E2 -9038.597} C_VEL
LIN {X 0,Y 439.381,Z 151.254,A -85,B 0,C 180,E1 -9041.256,E2 -9041.256} C_VEL
LIN {X 0,Y 439.398,Z 151.248,A -85,B 0,C 180,E1 -9044.73,E2 -9044.73} C_VEL
LIN {X 0,Y 439.382,Z 151.252,A -85,B 0,C 180,E1 -9047.794,E2 -9047.794} C_VEL
LIN {X 0,Y 439.358,Z 151.253,A -85,B 0,C 180,E1 -9050.22,E2 -9050.22} C_VEL
LIN {X 0,Y 439.373,Z 151.252,A -85,B 0,C 180,E1 -9053.713,E2 -9053.713} C_VEL
LIN {X 0,Y 439.373,Z 151.258,A -85,B 0,C 180,E1 -9057.054,E2 -9057.054} C_VEL
LIN {X 0,Y 439.372,Z 151.256,A -85,B 0,C 180,E1 -9060.274,E2 -9060.274} C_VEL
LIN {X 0,Y 439.376,Z 151.254,A -85,B 0,C 180,E1 -9063.393,E2 -9063.393} C_VEL
LIN {X 0,Y 439.418,Z 151.4,A -85,B 0,C 180,E1 -9063.757,E2 -9063.757} C_VEL
LIN {X 0,Y 441.779,Z 163.47,A -85,B 0,C 180,E1 -9066.316,E2 -9066.316} C_VEL
LIN {X 0,Y 441.834,Z 167.027,A -85,B 0,C 180,E1 -9067.024,E2 -9067.024} C_VEL
LIN {X 0,Y 440.872,Z 184.704,A -85,B 0,C 180,E1 -9070.442,E2 -9070.442} C_VEL
LIN {X 0,Y 440.497,Z 192.387,A -85,B 0,C 180,E1 -9071.873,E2 -9071.873} C_VEL
LIN {X 0,Y 444.066,Z 214.129,A -85,B 0,C 180,E1 -9072.384,E2 -9072.384} C_VEL
LIN {X 0,Y 443.286,Z 300.29,A -85,B 0,C 180,E1 -9073.803,E2 -9073.803} C_VEL
LIN {X 0,Y 442.877,Z 312.775,A -85,B 0,C 180,E1 -9074.172,E2 -9074.172} C_VEL
LIN {X 0,Y 442.326,Z 325.686,A -85,B 0,C 180,E1 -9074.743,E2 -9074.743} C_VEL
LIN {X 0,Y 441.654,Z 337.944,A -85,B 0,C 180,E1 -9075.485,E2 -9075.485} C_VEL
LIN {X 0,Y 441.011,Z 348.802,A -85,B 0,C 180,E1 -9076.339,E2 -9076.339} C_VEL
LIN {X 0,Y 440.409,Z 359.969,A -85,B 0,C 180,E1 -9077.442,E2 -9077.442} C_VEL
LIN {X 0,Y 439.873,Z 368.501,A -85,B 0,C 180,E1 -9078.48,E2 -9078.48} C_VEL
LIN {X 0,Y 439.355,Z 376.372,A -85,B 0,C 180,E1 -9079.633,E2 -9079.633} C_VEL
LIN {X 0,Y 438.921,Z 384.06,A -85,B 0,C 180,E1 -9081.018,E2 -9081.018} C_VEL
LIN {X 0,Y 438.582,Z 391.149,A -85,B 0,C 180,E1 -9082.635,E2 -9082.635} C_VEL
LIN {X 0,Y 438.385,Z 395.738,A -85,B 0,C 180,E1 -9083.978,E2 -9083.978} C_VEL
LIN {X 0,Y 438.34,Z 399.469,A -85,B 0,C 180,E1 -9085.402,E2 -9085.402} C_VEL
LIN {X 0,Y 438.259,Z 401.327,A -85,B 0,C 180,E1 -9086.322,E2 -9086.322} C_VEL
LIN {X 0,Y 438.334,Z 402.722,A -85,B 0,C 180,E1 -9087.243,E2 -9087.243} C_VEL
LIN {X 0,Y 438.231,Z 404.322,A -85,B 0,C 180,E1 -9089.081,E2 -9089.081} C_VEL
LIN {X 0,Y 438.23,Z 404.537,A -85,B 0,C 180,E1 -9090,E2 -9090} C_VEL
LIN {X 0,Y 438.278,Z 403.714,A -85,B 0,C 180,E1 -9091.838,E2 -9091.838} C_VEL
LIN {X 0,Y 438.334,Z 402.721,A -85,B 0,C 180,E1 -9092.757,E2 -9092.757} C_VEL
LIN {X 0,Y 438.259,Z 401.324,A -85,B 0,C 180,E1 -9093.678,E2 -9093.678} C_VEL
LIN {X 0,Y 438.383,Z 398.392,A -85,B 0,C 180,E1 -9095.059,E2 -9095.059} C_VEL
LIN {X 0,Y 438.449,Z 394.42,A -85,B 0,C 180,E1 -9096.442,E2 -9096.442} C_VEL
LIN {X 0,Y 438.684,Z 388.314,A -85,B 0,C 180,E1 -9098.058,E2 -9098.058} C_VEL
LIN {X 0,Y 439.043,Z 381.643,A -85,B 0,C 180,E1 -9099.444,E2 -9099.444} C_VEL
LIN {X 0,Y 439.498,Z 373.364,A -85,B 0,C 180,E1 -9100.83,E2 -9100.83} C_VEL
LIN {X 0,Y 440.097,Z 364.881,A -85,B 0,C 180,E1 -9101.982,E2 -9101.982} C_VEL
LIN {X 0,Y 440.714,Z 354.938,A -85,B 0,C 180,E1 -9103.081,E2 -9103.081} C_VEL
LIN {X 0,Y 441.284,Z 344.021,A -85,B 0,C 180,E1 -9104.056,E2 -9104.056} C_VEL
LIN {X 0,Y 441.923,Z 332.648,A -85,B 0,C 180,E1 -9104.859,E2 -9104.859} C_VEL
LIN {X 0,Y 442.49,Z 320.974,A -85,B 0,C 180,E1 -9105.488,E2 -9105.488} C_VEL
LIN {X 0,Y 443.021,Z 309.35,A -85,B 0,C 180,E1 -9105.941,E2 -9105.941} C_VEL
LIN {X 0,Y 443.372,Z 295.717,A -85,B 0,C 180,E1 -9106.282,E2 -9106.282} C_VEL
LIN {X 0,Y 444.002,Z 213.635,A -85,B 0,C 180,E1 -9107.621,E2 -9107.621} C_VEL
LIN {X 0,Y 440.489,Z 192.007,A -85,B 0,C 180,E1 -9108.155,E2 -9108.155} C_VEL
LIN {X 0,Y 441.339,Z 175.938,A -85,B 0,C 180,E1 -9111.24,E2 -9111.24} C_VEL
LIN {X 0,Y 441.914,Z 164.69,A -85,B 0,C 180,E1 -9113.427,E2 -9113.427} C_VEL
LIN {X 0,Y 439.836,Z 153.432,A -85,B 0,C 180,E1 -9115.798,E2 -9115.798} C_VEL
LIN {X 0,Y 439.4,Z 151.252,A -85,B 0,C 180,E1 -9116.302,E2 -9116.302} C_VEL
LIN {X 0,Y 439.39,Z 151.249,A -85,B 0,C 180,E1 -9118.675,E2 -9118.675} C_VEL
LIN {X 0,Y 439.363,Z 151.252,A -85,B 0,C 180,E1 -9122.029,E2 -9122.029} C_VEL
LIN {X 0,Y 439.393,Z 151.25,A -85,B 0,C 180,E1 -9125.34,E2 -9125.34} C_VEL
LIN {X 0,Y 439.368,Z 151.257,A -85,B 0,C 180,E1 -9128.596,E2 -9128.596} C_VEL
LIN {X 0,Y 439.37,Z 151.252,A -85,B 0,C 180,E1 -9131.254,E2 -9131.254} C_VEL
LIN {X 0,Y 439.398,Z 151.253,A -85,B 0,C 180,E1 -9134.729,E2 -9134.729} C_VEL
LIN {X 0,Y 439.384,Z 151.25,A -85,B 0,C 180,E1 -9137.794,E2 -9137.794} C_VEL
LIN {X 0,Y 439.388,Z 151.254,A -85,B 0,C 180,E1 -9140.223,E2 -9140.223} C_VEL
LIN {X 0,Y 439.372,Z 151.252,A -85,B 0,C 180,E1 -9143.712,E2 -9143.712} C_VEL
LIN {X 0,Y 439.372,Z 151.251,A -85,B 0,C 180,E1 -9147.054,E2 -9147.054} C_VEL
LIN {X 0,Y 439.376,Z 151.256,A -85,B 0,C 180,E1 -9150.274,E2 -9150.274} C_VEL
LIN {X 0,Y 439.382,Z 151.251,A -85,B 0,C 180,E1 -9153.393,E2 -9153.393} C_VEL
LIN {X 0,Y 439.383,Z 151.251,A -85,B 0,C 180,E1 -9156.429,E2 -9156.429} C_VEL
LIN {X 0,Y 439.387,Z 151.251,A -85,B 0,C 180,E1 -9159.397,E2 -9159.397} C_VEL
LIN {X 0,Y 439.425,Z 151.246,A -85,B 0,C 180,E1 -9162.309,E2 -9162.309} C_VEL
LIN {X 0,Y 439.447,Z 151.243,A -85,B 0,C 180,E1 -9165.174,E2 -9165.174} C_VEL
LIN {X 0,Y 439.483,Z 151.24,A -85,B 0,C 180,E1 -9168.001,E2 -9168.001} C_VEL
LIN {X 0,Y 439.547,Z 151.233,A -85,B 0,C 180,E1 -9171.726,E2 -9171.726} C_VEL
LIN {X 0,Y 439.617,Z 151.22,A -85,B 0,C 180,E1 -9174.496,E2 -9174.496} C_VEL
LIN {X 0,Y 439.634,Z 151.218,A -85,B 0,C 180,E1 -9178.168,E2 -9178.168} C_VEL
LIN {X 0,Y 439.762,Z 151.203,A -85,B 0,C 180,E1 -9180,E2 -9180} C_VEL
LIN {X 0,Y 439.655,Z 151.218,A -85,B 0,C 180,E1 -9182.749,E2 -9182.749} C_VEL
LIN {X 0,Y 439.583,Z 151.225,A -85,B 0,C 180,E1 -9186.514,E2 -9186.514} C_VEL
LIN {X 0,Y 439.498,Z 151.239,A -85,B 0,C 180,E1 -9189.202,E2 -9189.202} C_VEL
LIN {X 0,Y 439.465,Z 151.246,A -85,B 0,C 180,E1 -9192.938,E2 -9192.938} C_VEL
LIN {X 0,Y 439.447,Z 151.244,A -85,B 0,C 180,E1 -9196.349,E2 -9196.349} C_VEL
LIN {X 0,Y 439.403,Z 151.247,A -85,B 0,C 180,E1 -9199.626,E2 -9199.626} C_VEL
LIN {X 0,Y 439.365,Z 151.259,A -85,B 0,C 180,E1 -9202.576,E2 -9202.576} C_VEL
LIN {X 0,Y 439.405,Z 151.247,A -85,B 0,C 180,E1 -9205.585,E2 -9205.585} C_VEL
LIN {X 0,Y 439.417,Z 151.249,A -85,B 0,C 180,E1 -9208.674,E2 -9208.674} C_VEL
LIN {X 0,Y 439.37,Z 151.255,A -85,B 0,C 180,E1 -9212.031,E2 -9212.031} C_VEL
LIN {X 0,Y 439.395,Z 151.248,A -85,B 0,C 180,E1 -9215.341,E2 -9215.341} C_VEL
LIN {X 0,Y 439.379,Z 151.252,A -85,B 0,C 180,E1 -9218.596,E2 -9218.596} C_VEL
LIN {X 0,Y 439.389,Z 151.249,A -85,B 0,C 180,E1 -9221.257,E2 -9221.257} C_VEL
LIN {X 0,Y 439.404,Z 151.247,A -85,B 0,C 180,E1 -9224.729,E2 -9224.729} C_VEL
LIN {X 0,Y 439.397,Z 151.255,A -85,B 0,C 180,E1 -9227.796,E2 -9227.796} C_VEL
LIN {X 0,Y 439.396,Z 151.25,A -85,B 0,C 180,E1 -9230.224,E2 -9230.224} C_VEL
LIN {X 0,Y 439.375,Z 151.257,A -85,B 0,C 180,E1 -9233.713,E2 -9233.713} C_VEL
LIN {X 0,Y 439.373,Z 151.253,A -85,B 0,C 180,E1 -9237.054,E2 -9237.054} C_VEL
LIN {X 0,Y 439.384,Z 151.249,A -85,B 0,C 180,E1 -9240.274,E2 -9240.274} C_VEL
LIN {X 0,Y 439.431,Z 151.251,A -85,B 0,C 180,E1 -9243.396,E2 -9243.396} C_VEL
LIN {X 0,Y 439.431,Z 151.248,A -85,B 0,C 180,E1 -9246.931,E2 -9246.931} C_VEL
LIN {X 0,Y 439.453,Z 151.389,A -85,B 0,C 180,E1 -9247.119,E2 -9247.119} C_VEL
LIN {X 0,Y 441.139,Z 160.661,A -85,B 0,C 180,E1 -9249.239,E2 -9249.239} C_VEL
LIN {X 0,Y 440.73,Z 172.963,A -85,B 0,C 180,E1 -9251.835,E2 -9251.835} C_VEL
LIN {X 0,Y 440.706,Z 173.423,A -85,B 0,C 180,E1 -9251.931,E2 -9251.931} C_VEL
LIN {X 0,Y 444.292,Z 192.245,A -85,B 0,C 180,E1 -9252.401,E2 -9252.401} C_VEL
LIN {X 0,Y 443.398,Z 281.185,A -85,B 0,C 180,E1 -9253.867,E2 -9253.867} C_VEL
LIN {X 0,Y 442.997,Z 295.048,A -85,B 0,C 180,E1 -9254.295,E2 -9254.295} C_VEL
LIN {X 0,Y 442.896,Z 296.829,A -85,B 0,C 180,E1 -9254.362,E2 -9254.362} C_VEL
LIN {X 0,Y 442.138,Z 300.582,A -85,B 0,C 180,E1 -9254.501,E2 -9254.501} C_VEL
LIN {X 0,Y 439.173,Z 306.471,A -85,B 0,C 180,E1 -9254.692,E2 -9254.692} C_VEL
LIN {X 0,Y 436.128,Z 312.272,A -85,B 0,C 180,E1 -9254.92,E2 -9254.92} C_VEL
LIN {X 0,Y 435.26,Z 315.829,A -85,B 0,C 180,E1 -9255.126,E2 -9255.126} C_VEL
LIN {X 0,Y 434.66,Z 326.921,A -85,B 0,C 180,E1 -9255.964,E2 -9255.964} C_VEL
LIN {X 0,Y 434.053,Z 337.901,A -85,B 0,C 180,E1 -9257.017,E2 -9257.017} C_VEL
LIN {X 0,Y 433.286,Z 348.59,A -85,B 0,C 180,E1 -9258.302,E2 -9258.302} C_VEL
LIN {X 0,Y 432.745,Z 356.471,A -85,B 0,C 180,E1 -9259.473,E2 -9259.473} C_VEL
LIN {X 0,Y 432.228,Z 364.175,A -85,B 0,C 180,E1 -9260.878,E2 -9260.878} C_VEL
LIN {X 0,Y 431.785,Z 371.244,A -85,B 0,C 180,E1 -9262.518,E2 -9262.518} C_VEL
LIN {X 0,Y 431.598,Z 375.951,A -85,B 0,C 180,E1 -9263.924,E2 -9263.924} C_VEL
LIN {X 0,Y 431.346,Z 379.559,A -85,B 0,C 180,E1 -9265.327,E2 -9265.327} C_VEL
LIN {X 0,Y 431.321,Z 381.422,A -85,B 0,C 180,E1 -9266.263,E2 -9266.263} C_VEL
LIN {X 0,Y 431.331,Z 382.824,A -85,B 0,C 180,E1 -9267.198,E2 -9267.198} C_VEL
LIN {X 0,Y 431.173,Z 384.44,A -85,B 0,C 180,E1 -9269.066,E2 -9269.066} C_VEL
LIN {X 0,Y 431.147,Z 384.676,A -85,B 0,C 180,E1 -9270,E2 -9270} C_VEL
LIN {X 0,Y 431.173,Z 384.488,A -85,B 0,C 180,E1 -9270.934,E2 -9270.934} C_VEL
LIN {X 0,Y 431.33,Z 382.935,A -85,B 0,C 180,E1 -9272.802,E2 -9272.802} C_VEL
LIN {X 0,Y 431.316,Z 381.58,A -85,B 0,C 180,E1 -9273.737,E2 -9273.737} C_VEL
LIN {X 0,Y 431.422,Z 378.713,A -85,B 0,C 180,E1 -9275.14,E2 -9275.14} C_VEL
LIN {X 0,Y 431.619,Z 374.483,A -85,B 0,C 180,E1 -9276.656,E2 -9276.656} C_VEL
LIN {X 0,Y 431.875,Z 369.808,A -85,B 0,C 180,E1 -9277.951,E2 -9277.951} C_VEL
LIN {X 0,Y 432.295,Z 363.493,A -85,B 0,C 180,E1 -9279.356,E2 -9279.356} C_VEL
LIN {X 0,Y 432.826,Z 355.587,A -85,B 0,C 180,E1 -9280.762,E2 -9280.762} C_VEL
LIN {X 0,Y 433.361,Z 347.528,A -85,B 0,C 180,E1 -9281.933,E2 -9281.933} C_VEL
LIN {X 0,Y 434.095,Z 337.691,A -85,B 0,C 180,E1 -9283.1,E2 -9283.1} C_VEL
LIN {X 0,Y 434.723,Z 326.635,A -85,B 0,C 180,E1 -9284.153,E2 -9284.153} C_VEL
LIN {X 0,Y 435.279,Z 315.793,A -85,B 0,C 180,E1 -9284.971,E2 -9284.971} C_VEL
LIN {X 0,Y 435.907,Z 303.817,A -85,B 0,C 180,E1 -9285.667,E2 -9285.667} C_VEL
LIN {X 0,Y 436.379,Z 290.677,A -85,B 0,C 180,E1 -9286.22,E2 -9286.22} C_VEL
LIN {X 0,Y 436.699,Z 277.456,A -85,B 0,C 180,E1 -9286.568,E2 -9286.568} C_VEL
LIN {X 0,Y 437.483,Z 192.494,A -85,B 0,C 180,E1 -9287.977,E2 -9287.977} C_VEL
LIN {X 0,Y 433.776,Z 173.578,A -85,B 0,C 180,E1 -9288.466,E2 -9288.466} C_VEL
LIN {X 0,Y 434.277,Z 162.374,A -85,B 0,C 180,E1 -9290.856,E2 -9290.856} C_VEL
LIN {X 0,Y 432.358,Z 152.129,A -85,B 0,C 180,E1 -9293.247,E2 -9293.247} C_VEL
LIN {X 0,Y 432.401,Z 152.126,A -85,B 0,C 180,E1 -9296.627,E2 -9296.627} C_VEL
LIN {X 0,Y 432.344,Z 152.128,A -85,B 0,C 180,E1 -9299.187,E2 -9299.187} C_VEL
LIN {X 0,Y 432.323,Z 152.135,A -85,B 0,C 180,E1 -9302.443,E2 -9302.443} C_VEL
LIN {X 0,Y 432.344,Z 152.126,A -85,B 0,C 180,E1 -9305.631,E2 -9305.631} C_VEL
LIN {X 0,Y 432.339,Z 152.13,A -85,B 0,C 180,E1 -9308.714,E2 -9308.714} C_VEL
LIN {X 0,Y 432.334,Z 152.13,A -85,B 0,C 180,E1 -9311.797,E2 -9311.797} C_VEL
LIN {X 0,Y 432.334,Z 152.133,A -85,B 0,C 180,E1 -9314.347,E2 -9314.347} C_VEL
LIN {X 0,Y 432.321,Z 152.129,A -85,B 0,C 180,E1 -9317.015,E2 -9317.015} C_VEL
LIN {X 0,Y 432.333,Z 152.132,A -85,B 0,C 180,E1 -9319.821,E2 -9319.821} C_VEL
LIN {X 0,Y 432.306,Z 152.131,A -85,B 0,C 180,E1 -9323.022,E2 -9323.022} C_VEL
LIN {X 0,Y 432.359,Z 152.13,A -85,B 0,C 180,E1 -9325.996,E2 -9325.996} C_VEL
LIN {X 0,Y 432.347,Z 152.13,A -85,B 0,C 180,E1 -9329.489,E2 -9329.489} C_VEL
LIN {X 0,Y 432.391,Z 152.121,A -85,B 0,C 180,E1 -9332.928,E2 -9332.928} C_VEL
LIN {X 0,Y 432.371,Z 152.125,A -85,B 0,C 180,E1 -9336.023,E2 -9336.023} C_VEL
LIN {X 0,Y 432.35,Z 152.128,A -85,B 0,C 180,E1 -9339.046,E2 -9339.046} C_VEL
LIN {X 0,Y 432.378,Z 152.123,A -85,B 0,C 180,E1 -9342.011,E2 -9342.011} C_VEL
LIN {X 0,Y 432.395,Z 152.123,A -85,B 0,C 180,E1 -9344.926,E2 -9344.926} C_VEL
LIN {X 0,Y 432.459,Z 152.113,A -85,B 0,C 180,E1 -9347.803,E2 -9347.803} C_VEL
LIN {X 0,Y 432.491,Z 152.11,A -85,B 0,C 180,E1 -9351.59,E2 -9351.59} C_VEL
LIN {X 0,Y 432.593,Z 152.097,A -85,B 0,C 180,E1 -9354.406,E2 -9354.406} C_VEL
LIN {X 0,Y 432.605,Z 152.094,A -85,B 0,C 180,E1 -9358.138,E2 -9358.138} C_VEL
LIN {X 0,Y 432.731,Z 152.078,A -85,B 0,C 180,E1 -9360,E2 -9360} C_VEL
LIN {X 0,Y 432.603,Z 152.101,A -85,B 0,C 180,E1 -9362.794,E2 -9362.794} C_VEL
LIN {X 0,Y 432.564,Z 152.105,A -85,B 0,C 180,E1 -9366.53,E2 -9366.53} C_VEL
LIN {X 0,Y 432.441,Z 152.114,A -85,B 0,C 180,E1 -9369.353,E2 -9369.353} C_VEL
LIN {X 0,Y 432.43,Z 152.119,A -85,B 0,C 180,E1 -9372.804,E2 -9372.804} C_VEL
LIN {X 0,Y 432.411,Z 152.123,A -85,B 0,C 180,E1 -9376.479,E2 -9376.479} C_VEL
LIN {X 0,Y 432.338,Z 152.131,A -85,B 0,C 180,E1 -9379.961,E2 -9379.961} C_VEL
LIN {X 0,Y 432.317,Z 152.13,A -85,B 0,C 180,E1 -9382.964,E2 -9382.964} C_VEL
LIN {X 0,Y 432.36,Z 152.132,A -85,B 0,C 180,E1 -9386.033,E2 -9386.033} C_VEL
LIN {X 0,Y 432.342,Z 152.127,A -85,B 0,C 180,E1 -9389.188,E2 -9389.188} C_VEL
LIN {X 0,Y 432.322,Z 152.13,A -85,B 0,C 180,E1 -9392.443,E2 -9392.443} C_VEL
LIN {X 0,Y 432.342,Z 152.133,A -85,B 0,C 180,E1 -9395.632,E2 -9395.632} C_VEL
LIN {X 0,Y 432.332,Z 152.128,A -85,B 0,C 180,E1 -9398.713,E2 -9398.713} C_VEL
LIN {X 0,Y 432.323,Z 152.133,A -85,B 0,C 180,E1 -9401.798,E2 -9401.798} C_VEL
LIN {X 0,Y 432.333,Z 152.128,A -85,B 0,C 180,E1 -9404.348,E2 -9404.348} C_VEL
LIN {X 0,Y 432.316,Z 152.133,A -85,B 0,C 180,E1 -9407.017,E2 -9407.017} C_VEL
LIN {X 0,Y 432.308,Z 152.132,A -85,B 0,C 180,E1 -9409.825,E2 -9409.825} C_VEL
LIN {X 0,Y 432.306,Z 152.136,A -85,B 0,C 180,E1 -9413.022,E2 -9413.022} C_VEL
LIN {X 0,Y 432.358,Z 152.125,A -85,B 0,C 180,E1 -9415.997,E2 -9415.997} C_VEL
LIN {X 0,Y 432.346,Z 152.133,A -85,B 0,C 180,E1 -9419.49,E2 -9419.49} C_VEL
LIN {X 0,Y 432.339,Z 152.128,A -85,B 0,C 180,E1 -9421.874,E2 -9421.874} C_VEL
LIN {X 0,Y 432.356,Z 152.151,A -85,B 0,C 180,E1 -9423.485,E2 -9423.485} C_VEL
LIN {X 0,Y 434.794,Z 164.558,A -85,B 0,C 180,E1 -9426.165,E2 -9426.165} C_VEL
LIN {X 0,Y 434.972,Z 167.316,A -85,B 0,C 180,E1 -9426.731,E2 -9426.731} C_VEL
LIN {X 0,Y 433.895,Z 185.789,A -85,B 0,C 180,E1 -9430.361,E2 -9430.361} C_VEL
LIN {X 0,Y 433.544,Z 191.992,A -85,B 0,C 180,E1 -9431.567,E2 -9431.567} C_VEL
LIN {X 0,Y 437.286,Z 215.217,A -85,B 0,C 180,E1 -9432.123,E2 -9432.123} C_VEL
LIN {X 0,Y 436.486,Z 300.14,A -85,B 0,C 180,E1 -9433.544,E2 -9433.544} C_VEL
LIN {X 0,Y 436.056,Z 312.621,A -85,B 0,C 180,E1 -9433.918,E2 -9433.918} C_VEL
LIN {X 0,Y 435.469,Z 325.53,A -85,B 0,C 180,E1 -9434.496,E2 -9434.496} C_VEL
LIN {X 0,Y 434.773,Z 337.785,A -85,B 0,C 180,E1 -9435.251,E2 -9435.251} C_VEL
LIN {X 0,Y 434.071,Z 349.039,A -85,B 0,C 180,E1 -9436.153,E2 -9436.153} C_VEL
LIN {X 0,Y 433.453,Z 359.809,A -85,B 0,C 180,E1 -9437.237,E2 -9437.237} C_VEL
LIN {X 0,Y 432.895,Z 368.34,A -85,B 0,C 180,E1 -9438.291,E2 -9438.291} C_VEL
LIN {X 0,Y 432.333,Z 376.211,A -85,B 0,C 180,E1 -9439.463,E2 -9439.463} C_VEL
LIN {X 0,Y 431.862,Z 383.898,A -85,B 0,C 180,E1 -9440.87,E2 -9440.87} C_VEL
LIN {X 0,Y 431.516,Z 390.987,A -85,B 0,C 180,E1 -9442.513,E2 -9442.513} C_VEL
LIN {X 0,Y 431.285,Z 396.005,A -85,B 0,C 180,E1 -9444.019,E2 -9444.019} C_VEL
LIN {X 0,Y 431.27,Z 399.308,A -85,B 0,C 180,E1 -9445.326,E2 -9445.326} C_VEL
LIN {X 0,Y 431.167,Z 401.165,A -85,B 0,C 180,E1 -9446.262,E2 -9446.262} C_VEL
LIN {X 0,Y 431.228,Z 402.56,A -85,B 0,C 180,E1 -9447.198,E2 -9447.198} C_VEL
LIN {X 0,Y 431.202,Z 403.554,A -85,B 0,C 180,E1 -9448.132,E2 -9448.132} C_VEL
LIN {X 0,Y 431.145,Z 404.375,A -85,B 0,C 180,E1 -9450,E2 -9450} C_VEL
LIN {X 0,Y 431.202,Z 403.552,A -85,B 0,C 180,E1 -9451.868,E2 -9451.868} C_VEL
LIN {X 0,Y 431.228,Z 402.558,A -85,B 0,C 180,E1 -9452.803,E2 -9452.803} C_VEL
LIN {X 0,Y 431.167,Z 401.161,A -85,B 0,C 180,E1 -9453.738,E2 -9453.738} C_VEL
LIN {X 0,Y 431.294,Z 398.229,A -85,B 0,C 180,E1 -9455.142,E2 -9455.142} C_VEL
LIN {X 0,Y 431.377,Z 394.257,A -85,B 0,C 180,E1 -9456.549,E2 -9456.549} C_VEL
LIN {X 0,Y 431.625,Z 388.15,A -85,B 0,C 180,E1 -9458.191,E2 -9458.191} C_VEL
LIN {X 0,Y 431.993,Z 381.478,A -85,B 0,C 180,E1 -9459.599,E2 -9459.599} C_VEL
LIN {X 0,Y 432.505,Z 373.2,A -85,B 0,C 180,E1 -9461.007,E2 -9461.007} C_VEL
LIN {X 0,Y 433.14,Z 364.716,A -85,B 0,C 180,E1 -9462.177,E2 -9462.177} C_VEL
LIN {X 0,Y 433.757,Z 353.829,A -85,B 0,C 180,E1 -9463.39,E2 -9463.39} C_VEL
LIN {X 0,Y 434.47,Z 342.426,A -85,B 0,C 180,E1 -9464.401,E2 -9464.401} C_VEL
LIN {X 0,Y 435.175,Z 330.555,A -85,B 0,C 180,E1 -9465.215,E2 -9465.215} C_VEL
LIN {X 0,Y 435.728,Z 318.2,A -85,B 0,C 180,E1 -9465.854,E2 -9465.854} C_VEL
LIN {X 0,Y 436.323,Z 305.516,A -85,B 0,C 180,E1 -9466.312,E2 -9466.312} C_VEL
LIN {X 0,Y 436.595,Z 292.221,A -85,B 0,C 180,E1 -9466.602,E2 -9466.602} C_VEL
LIN {X 0,Y 437.29,Z 215.206,A -85,B 0,C 180,E1 -9467.871,E2 -9467.871} C_VEL
LIN {X 0,Y 433.534,Z 191.974,A -85,B 0,C 180,E1 -9468.43,E2 -9468.43} C_VEL
LIN {X 0,Y 434.431,Z 175.773,A -85,B 0,C 180,E1 -9471.595,E2 -9471.595} C_VEL
LIN {X 0,Y 434.971,Z 165.777,A -85,B 0,C 180,E1 -9473.571,E2 -9473.571} C_VEL
LIN {X 0,Y 432.842,Z 154.447,A -85,B 0,C 180,E1 -9476.001,E2 -9476.001} C_VEL
LIN {X 0,Y 432.348,Z 152.13,A -85,B 0,C 180,E1 -9476.513,E2 -9476.513} C_VEL
LIN {X 0,Y 432.327,Z 152.134,A -85,B 0,C 180,E1 -9479.189,E2 -9479.189} C_VEL
LIN {X 0,Y 432.32,Z 152.131,A -85,B 0,C 180,E1 -9482.443,E2 -9482.443} C_VEL
LIN {X 0,Y 432.338,Z 152.127,A -85,B 0,C 180,E1 -9485.818,E2 -9485.818} C_VEL
LIN {X 0,Y 432.33,Z 152.135,A -85,B 0,C 180,E1 -9488.712,E2 -9488.712} C_VEL
LIN {X 0,Y 432.32,Z 152.129,A -85,B 0,C 180,E1 -9491.799,E2 -9491.799} C_VEL
LIN {X 0,Y 432.334,Z 152.132,A -85,B 0,C 180,E1 -9494.347,E2 -9494.347} C_VEL
LIN {X 0,Y 432.316,Z 152.132,A -85,B 0,C 180,E1 -9497.016,E2 -9497.016} C_VEL
LIN {X 0,Y 432.331,Z 152.129,A -85,B 0,C 180,E1 -9499.821,E2 -9499.821} C_VEL
LIN {X 0,Y 432.304,Z 152.132,A -85,B 0,C 180,E1 -9503.022,E2 -9503.022} C_VEL
LIN {X 0,Y 432.359,Z 152.129,A -85,B 0,C 180,E1 -9505.996,E2 -9505.996} C_VEL
LIN {X 0,Y 432.346,Z 152.127,A -85,B 0,C 180,E1 -9509.49,E2 -9509.49} C_VEL
LIN {X 0,Y 432.347,Z 152.131,A -85,B 0,C 180,E1 -9511.874,E2 -9511.874} C_VEL
LIN {X 0,Y 432.378,Z 152.125,A -85,B 0,C 180,E1 -9515.538,E2 -9515.538} C_VEL
LIN {X 0,Y 432.349,Z 152.126,A -85,B 0,C 180,E1 -9519.046,E2 -9519.046} C_VEL
LIN {X 0,Y 432.373,Z 152.127,A -85,B 0,C 180,E1 -9522.011,E2 -9522.011} C_VEL
LIN {X 0,Y 432.395,Z 152.12,A -85,B 0,C 180,E1 -9524.926,E2 -9524.926} C_VEL
LIN {X 0,Y 432.459,Z 152.117,A -85,B 0,C 180,E1 -9527.803,E2 -9527.803} C_VEL
LIN {X 0,Y 432.491,Z 152.114,A -85,B 0,C 180,E1 -9531.59,E2 -9531.59} C_VEL
LIN {X 0,Y 432.594,Z 152.095,A -85,B 0,C 180,E1 -9534.406,E2 -9534.406} C_VEL
LIN {X 0,Y 432.604,Z 152.094,A -85,B 0,C 180,E1 -9538.138,E2 -9538.138} C_VEL
LIN {X 0,Y 432.732,Z 152.078,A -85,B 0,C 180,E1 -9540,E2 -9540} C_VEL
LIN {X 0,Y 432.604,Z 152.097,A -85,B 0,C 180,E1 -9542.794,E2 -9542.794} C_VEL
LIN {X 0,Y 432.544,Z 152.103,A -85,B 0,C 180,E1 -9546.516,E2 -9546.516} C_VEL
LIN {X 0,Y 432.441,Z 152.117,A -85,B 0,C 180,E1 -9549.353,E2 -9549.353} C_VEL
LIN {X 0,Y 432.431,Z 152.122,A -85,B 0,C 180,E1 -9552.804,E2 -9552.804} C_VEL
LIN {X 0,Y 432.413,Z 152.122,A -85,B 0,C 180,E1 -9556.479,E2 -9556.479} C_VEL
LIN {X 0,Y 432.339,Z 152.128,A -85,B 0,C 180,E1 -9559.961,E2 -9559.961} C_VEL
LIN {X 0,Y 432.319,Z 152.132,A -85,B 0,C 180,E1 -9562.964,E2 -9562.964} C_VEL
LIN {X 0,Y 432.364,Z 152.126,A -85,B 0,C 180,E1 -9566.033,E2 -9566.033} C_VEL
LIN {X 0,Y 432.343,Z 152.127,A -85,B 0,C 180,E1 -9569.188,E2 -9569.188} C_VEL
LIN {X 0,Y 432.323,Z 152.134,A -85,B 0,C 180,E1 -9572.443,E2 -9572.443} C_VEL
LIN {X 0,Y 432.344,Z 152.128,A -85,B 0,C 180,E1 -9575.632,E2 -9575.632} C_VEL
LIN {X 0,Y 432.347,Z 152.126,A -85,B 0,C 180,E1 -9579.343,E2 -9579.343} C_VEL
LIN {X 0,Y 432.335,Z 152.133,A -85,B 0,C 180,E1 -9581.797,E2 -9581.797} C_VEL
LIN {X 0,Y 432.338,Z 152.129,A -85,B 0,C 180,E1 -9584.347,E2 -9584.347} C_VEL
LIN {X 0,Y 432.321,Z 152.129,A -85,B 0,C 180,E1 -9587.016,E2 -9587.016} C_VEL
LIN {X 0,Y 432.335,Z 152.134,A -85,B 0,C 180,E1 -9589.821,E2 -9589.821} C_VEL
LIN {X 0,Y 432.307,Z 152.132,A -85,B 0,C 180,E1 -9593.022,E2 -9593.022} C_VEL
LIN {X 0,Y 432.359,Z 152.127,A -85,B 0,C 180,E1 -9595.997,E2 -9595.997} C_VEL
LIN {X 0,Y 432.349,Z 152.133,A -85,B 0,C 180,E1 -9599.49,E2 -9599.49} C_VEL
LIN {X 0,Y 432.393,Z 152.123,A -85,B 0,C 180,E1 -9602.928,E2 -9602.928} C_VEL
LIN {X 0,Y 432.378,Z 152.125,A -85,B 0,C 180,E1 -9606.532,E2 -9606.532} C_VEL
LIN {X 0,Y 432.423,Z 152.353,A -85,B 0,C 180,E1 -9606.915,E2 -9606.915} C_VEL
LIN {X 0,Y 434.18,Z 161.93,A -85,B 0,C 180,E1 -9609.139,E2 -9609.139} C_VEL
LIN {X 0,Y 433.789,Z 173.562,A -85,B 0,C 180,E1 -9611.628,E2 -9611.628} C_VEL
LIN {X 0,Y 437.516,Z 192.788,A -85,B 0,C 180,E1 -9612.126,E2 -9612.126} C_VEL
LIN {X 0,Y 436.601,Z 281.363,A -85,B 0,C 180,E1 -9613.608,E2 -9613.608} C_VEL
LIN {X 0,Y 436.188,Z 295.221,A -85,B 0,C 180,E1 -9614.043,E2 -9614.043} C_VEL
LIN {X 0,Y 435.653,Z 307.626,A -85,B 0,C 180,E1 -9614.623,E2 -9614.623} C_VEL
LIN {X 0,Y 435.26,Z 315.829,A -85,B 0,C 180,E1 -9615.126,E2 -9615.126} C_VEL
LIN {X 0,Y 434.377,Z 319.383,A -85,B 0,C 180,E1 -9615.344,E2 -9615.344} C_VEL
LIN {X 0,Y 428.241,Z 330.238,A -85,B 0,C 180,E1 -9616.036,E2 -9616.036} C_VEL
LIN {X 0,Y 427.466,Z 333.467,A -85,B 0,C 180,E1 -9616.327,E2 -9616.327} C_VEL
LIN {X 0,Y 426.796,Z 343.221,A -85,B 0,C 180,E1 -9617.397,E2 -9617.397} C_VEL
LIN {X 0,Y 426.075,Z 352.075,A -85,B 0,C 180,E1 -9618.584,E2 -9618.584} C_VEL
LIN {X 0,Y 425.466,Z 360.711,A -85,B 0,C 180,E1 -9620.012,E2 -9620.012} C_VEL
LIN {X 0,Y 424.972,Z 367.595,A -85,B 0,C 180,E1 -9621.44,E2 -9621.44} C_VEL
LIN {X 0,Y 424.631,Z 373.266,A -85,B 0,C 180,E1 -9622.917,E2 -9622.917} C_VEL
LIN {X 0,Y 424.456,Z 377.431,A -85,B 0,C 180,E1 -9624.298,E2 -9624.298} C_VEL
LIN {X 0,Y 424.28,Z 379.722,A -85,B 0,C 180,E1 -9625.249,E2 -9625.249} C_VEL
LIN {X 0,Y 424.225,Z 381.585,A -85,B 0,C 180,E1 -9626.2,E2 -9626.2} C_VEL
LIN {X 0,Y 424.244,Z 382.987,A -85,B 0,C 180,E1 -9627.151,E2 -9627.151} C_VEL
LIN {X 0,Y 424.093,Z 384.602,A -85,B 0,C 180,E1 -9629.05,E2 -9629.05} C_VEL
LIN {X 0,Y 424.065,Z 384.838,A -85,B 0,C 180,E1 -9630,E2 -9630} C_VEL
LIN {X 0,Y 424.093,Z 384.65,A -85,B 0,C 180,E1 -9630.949,E2 -9630.949} C_VEL
LIN {X 0,Y 424.243,Z 383.096,A -85,B 0,C 180,E1 -9632.849,E2 -9632.849} C_VEL
LIN {X 0,Y 424.22,Z 381.741,A -85,B 0,C 180,E1 -9633.8,E2 -9633.8} C_VEL
LIN {X 0,Y 424.365,Z 378.873,A -85,B 0,C 180,E1 -9635.226,E2 -9635.226} C_VEL
LIN {X 0,Y 424.542,Z 374.985,A -85,B 0,C 180,E1 -9636.654,E2 -9636.654} C_VEL
LIN {X 0,Y 424.821,Z 369.969,A -85,B 0,C 180,E1 -9638.084,E2 -9638.084} C_VEL
LIN {X 0,Y 425.299,Z 363.653,A -85,B 0,C 180,E1 -9639.512,E2 -9639.512} C_VEL
LIN {X 0,Y 425.828,Z 355.747,A -85,B 0,C 180,E1 -9640.941,E2 -9640.941} C_VEL
LIN {X 0,Y 426.418,Z 347.687,A -85,B 0,C 180,E1 -9642.13,E2 -9642.13} C_VEL
LIN {X 0,Y 427.182,Z 337.85,A -85,B 0,C 180,E1 -9643.316,E2 -9643.316} C_VEL
LIN {X 0,Y 427.838,Z 326.792,A -85,B 0,C 180,E1 -9644.386,E2 -9644.386} C_VEL
LIN {X 0,Y 428.437,Z 315.948,A -85,B 0,C 180,E1 -9645.216,E2 -9645.216} C_VEL
LIN {X 0,Y 429.075,Z 303.971,A -85,B 0,C 180,E1 -9645.923,E2 -9645.923} C_VEL
LIN {X 0,Y 429.577,Z 290.826,A -85,B 0,C 180,E1 -9646.484,E2 -9646.484} C_VEL
LIN {X 0,Y 429.915,Z 277.595,A -85,B 0,C 180,E1 -9646.837,E2 -9646.837} C_VEL
LIN {X 0,Y 430.679,Z 193.072,A -85,B 0,C 180,E1 -9648.263,E2 -9648.263} C_VEL
LIN {X 0,Y 426.893,Z 173.647,A -85,B 0,C 180,E1 -9648.793,E2 -9648.793} C_VEL
LIN {X 0,Y 427.345,Z 163.764,A -85,B 0,C 180,E1 -9650.933,E2 -9650.933} C_VEL
LIN {X 0,Y 425.332,Z 153.005,A -85,B 0,C 180,E1 -9653.492,E2 -9653.492} C_VEL
LIN {X 0,Y 425.35,Z 153.004,A -85,B 0,C 180,E1 -9656.844,E2 -9656.844} C_VEL
LIN {X 0,Y 425.292,Z 153.005,A -85,B 0,C 180,E1 -9659.719,E2 -9659.719} C_VEL
LIN {X 0,Y 425.283,Z 153.008,A -85,B 0,C 180,E1 -9663.048,E2 -9663.048} C_VEL
LIN {X 0,Y 425.282,Z 153.008,A -85,B 0,C 180,E1 -9665.928,E2 -9665.928} C_VEL
LIN {X 0,Y 425.282,Z 153.007,A -85,B 0,C 180,E1 -9669.04,E2 -9669.04} C_VEL
LIN {X 0,Y 425.29,Z 153.008,A -85,B 0,C 180,E1 -9671.958,E2 -9671.958} C_VEL
LIN {X 0,Y 425.288,Z 153.005,A -85,B 0,C 180,E1 -9675.282,E2 -9675.282} C_VEL
LIN {X 0,Y 425.274,Z 153.009,A -85,B 0,C 180,E1 -9678.621,E2 -9678.621} C_VEL
LIN {X 0,Y 425.306,Z 153.003,A -85,B 0,C 180,E1 -9681.102,E2 -9681.102} C_VEL
LIN {X 0,Y 425.299,Z 153.004,A -85,B 0,C 180,E1 -9684.664,E2 -9684.664} C_VEL
LIN {X 0,Y 425.265,Z 153.012,A -85,B 0,C 180,E1 -9688.073,E2 -9688.073} C_VEL
LIN {X 0,Y 425.331,Z 153.003,A -85,B 0,C 180,E1 -9691.368,E2 -9691.368} C_VEL
LIN {X 0,Y 425.295,Z 153.004,A -85,B 0,C 180,E1 -9694.554,E2 -9694.554} C_VEL
LIN {X 0,Y 425.287,Z 153.011,A -85,B 0,C 180,E1 -9697.661,E2 -9697.661} C_VEL
LIN {X 0,Y 425.362,Z 152.997,A -85,B 0,C 180,E1 -9700.704,E2 -9700.704} C_VEL
LIN {X 0,Y 425.388,Z 152.996,A -85,B 0,C 180,E1 -9703.688,E2 -9703.688} C_VEL
LIN {X 0,Y 425.411,Z 152.993,A -85,B 0,C 180,E1 -9707.598,E2 -9707.598} C_VEL
LIN {X 0,Y 425.442,Z 152.989,A -85,B 0,C 180,E1 -9711.45,E2 -9711.45} C_VEL
LIN {X 0,Y 425.549,Z 152.974,A -85,B 0,C 180,E1 -9714.313,E2 -9714.313} C_VEL
LIN {X 0,Y 425.575,Z 152.97,A -85,B 0,C 180,E1 -9718.107,E2 -9718.107} C_VEL
LIN {X 0,Y 425.701,Z 152.954,A -85,B 0,C 180,E1 -9720,E2 -9720} C_VEL
LIN {X 0,Y 425.555,Z 152.978,A -85,B 0,C 180,E1 -9722.84,E2 -9722.84} C_VEL
LIN {X 0,Y 425.522,Z 152.983,A -85,B 0,C 180,E1 -9726.639,E2 -9726.639} C_VEL
LIN {X 0,Y 425.399,Z 152.991,A -85,B 0,C 180,E1 -9729.509,E2 -9729.509} C_VEL
LIN {X 0,Y 425.392,Z 152.994,A -85,B 0,C 180,E1 -9732.904,E2 -9732.904} C_VEL
LIN {X 0,Y 425.36,Z 153,A -85,B 0,C 180,E1 -9736.605,E2 -9736.605} C_VEL
LIN {X 0,Y 425.327,Z 153.002,A -85,B 0,C 180,E1 -9739.636,E2 -9739.636} C_VEL
LIN {X 0,Y 425.287,Z 153.01,A -85,B 0,C 180,E1 -9742.339,E2 -9742.339} C_VEL
LIN {X 0,Y 425.29,Z 153.006,A -85,B 0,C 180,E1 -9745.446,E2 -9745.446} C_VEL
LIN {X 0,Y 425.347,Z 153,A -85,B 0,C 180,E1 -9747.558,E2 -9747.558} C_VEL
LIN {X 0,Y 425.287,Z 153.005,A -85,B 0,C 180,E1 -9750.816,E2 -9750.816} C_VEL
LIN {X 0,Y 425.31,Z 153.004,A -85,B 0,C 180,E1 -9754.288,E2 -9754.288} C_VEL
LIN {X 0,Y 425.276,Z 153.014,A -85,B 0,C 180,E1 -9757.695,E2 -9757.695} C_VEL
LIN {X 0,Y 425.275,Z 153.007,A -85,B 0,C 180,E1 -9760.52,E2 -9760.52} C_VEL
LIN {X 0,Y 425.26,Z 153.011,A -85,B 0,C 180,E1 -9763.956,E2 -9763.956} C_VEL
LIN {X 0,Y 425.269,Z 153.015,A -85,B 0,C 180,E1 -9767.346,E2 -9767.346} C_VEL
LIN {X 0,Y 425.265,Z 153.012,A -85,B 0,C 180,E1 -9770.962,E2 -9770.962} C_VEL
LIN {X 0,Y 425.282,Z 153.006,A -85,B 0,C 180,E1 -9774.072,E2 -9774.072} C_VEL
LIN {X 0,Y 425.282,Z 153.012,A -85,B 0,C 180,E1 -9776.952,E2 -9776.952} C_VEL
LIN {X 0,Y 425.284,Z 153.011,A -85,B 0,C 180,E1 -9780.28,E2 -9780.28} C_VEL
LIN {X 0,Y 425.31,Z 153.099,A -85,B 0,C 180,E1 -9783.246,E2 -9783.246} C_VEL
LIN {X 0,Y 427.804,Z 165.645,A -85,B 0,C 180,E1 -9786.009,E2 -9786.009} C_VEL
LIN {X 0,Y 427.926,Z 169.879,A -85,B 0,C 180,E1 -9786.884,E2 -9786.884} C_VEL
LIN {X 0,Y 426.864,Z 188.118,A -85,B 0,C 180,E1 -9790.525,E2 -9790.525} C_VEL
LIN {X 0,Y 426.595,Z 191.828,A -85,B 0,C 180,E1 -9791.256,E2 -9791.256} C_VEL
LIN {X 0,Y 430.548,Z 216.074,A -85,B 0,C 180,E1 -9791.85,E2 -9791.85} C_VEL
LIN {X 0,Y 429.698,Z 299.991,A -85,B 0,C 180,E1 -9793.276,E2 -9793.276} C_VEL
LIN {X 0,Y 429.234,Z 312.466,A -85,B 0,C 180,E1 -9793.655,E2 -9793.655} C_VEL
LIN {X 0,Y 428.616,Z 325.373,A -85,B 0,C 180,E1 -9794.242,E2 -9794.242} C_VEL
LIN {X 0,Y 427.913,Z 337.627,A -85,B 0,C 180,E1 -9795.009,E2 -9795.009} C_VEL
LIN {X 0,Y 427.145,Z 348.784,A -85,B 0,C 180,E1 -9795.915,E2 -9795.915} C_VEL
LIN {X 0,Y 426.48,Z 359.649,A -85,B 0,C 180,E1 -9797.025,E2 -9797.025} C_VEL
LIN {X 0,Y 425.921,Z 368.18,A -85,B 0,C 180,E1 -9798.097,E2 -9798.097} C_VEL
LIN {X 0,Y 425.301,Z 376.049,A -85,B 0,C 180,E1 -9799.286,E2 -9799.286} C_VEL
LIN {X 0,Y 424.819,Z 383.737,A -85,B 0,C 180,E1 -9800.718,E2 -9800.718} C_VEL
LIN {X 0,Y 424.432,Z 390.825,A -85,B 0,C 180,E1 -9802.388,E2 -9802.388} C_VEL
LIN {X 0,Y 424.244,Z 395.185,A -85,B 0,C 180,E1 -9803.7,E2 -9803.7} C_VEL
LIN {X 0,Y 424.199,Z 399.146,A -85,B 0,C 180,E1 -9805.248,E2 -9805.248} C_VEL
LIN {X 0,Y 424.081,Z 401.003,A -85,B 0,C 180,E1 -9806.199,E2 -9806.199} C_VEL
LIN {X 0,Y 424.122,Z 402.398,A -85,B 0,C 180,E1 -9807.151,E2 -9807.151} C_VEL
LIN {X 0,Y 424.128,Z 403.393,A -85,B 0,C 180,E1 -9808.101,E2 -9808.101} C_VEL
LIN {X 0,Y 424.063,Z 404.214,A -85,B 0,C 180,E1 -9810,E2 -9810} C_VEL
LIN {X 0,Y 424.128,Z 403.39,A -85,B 0,C 180,E1 -9811.899,E2 -9811.899} C_VEL
LIN {X 0,Y 424.122,Z 402.395,A -85,B 0,C 180,E1 -9812.849,E2 -9812.849} C_VEL
LIN {X 0,Y 424.081,Z 400.998,A -85,B 0,C 180,E1 -9813.801,E2 -9813.801} C_VEL
LIN {X 0,Y 424.207,Z 398.065,A -85,B 0,C 180,E1 -9815.228,E2 -9815.228} C_VEL
LIN {X 0,Y 424.301,Z 394.093,A -85,B 0,C 180,E1 -9816.658,E2 -9816.658} C_VEL
LIN {X 0,Y 424.581,Z 387.986,A -85,B 0,C 180,E1 -9818.328,E2 -9818.328} C_VEL
LIN {X 0,Y 424.95,Z 381.313,A -85,B 0,C 180,E1 -9819.76,E2 -9819.76} C_VEL
LIN {X 0,Y 425.493,Z 373.034,A -85,B 0,C 180,E1 -9821.191,E2 -9821.191} C_VEL
LIN {X 0,Y 426.191,Z 364.551,A -85,B 0,C 180,E1 -9822.379,E2 -9822.379} C_VEL
LIN {X 0,Y 426.786,Z 354.446,A -85,B 0,C 180,E1 -9823.532,E2 -9823.532} C_VEL
LIN {X 0,Y 427.472,Z 343.688,A -85,B 0,C 180,E1 -9824.52,E2 -9824.52} C_VEL
LIN {X 0,Y 428.216,Z 332.315,A -85,B 0,C 180,E1 -9825.346,E2 -9825.346} C_VEL
LIN {X 0,Y 428.817,Z 320.636,A -85,B 0,C 180,E1 -9825.994,E2 -9825.994} C_VEL
LIN {X 0,Y 429.429,Z 308.091,A -85,B 0,C 180,E1 -9826.49,E2 -9826.49} C_VEL
LIN {X 0,Y 429.744,Z 295.361,A -85,B 0,C 180,E1 -9826.814,E2 -9826.814} C_VEL
LIN {X 0,Y 430.419,Z 215.109,A -85,B 0,C 180,E1 -9828.165,E2 -9828.165} C_VEL
LIN {X 0,Y 426.597,Z 191.74,A -85,B 0,C 180,E1 -9828.754,E2 -9828.754} C_VEL
LIN {X 0,Y 427.686,Z 174.361,A -85,B 0,C 180,E1 -9832.207,E2 -9832.207} C_VEL
LIN {X 0,Y 428.016,Z 166.86,A -85,B 0,C 180,E1 -9833.721,E2 -9833.721} C_VEL
LIN {X 0,Y 425.555,Z 154.271,A -85,B 0,C 180,E1 -9836.481,E2 -9836.481} C_VEL
LIN {X 0,Y 425.273,Z 153.011,A -85,B 0,C 180,E1 -9836.824,E2 -9836.824} C_VEL
LIN {X 0,Y 425.282,Z 153.005,A -85,B 0,C 180,E1 -9839.72,E2 -9839.72} C_VEL
LIN {X 0,Y 425.269,Z 153.013,A -85,B 0,C 180,E1 -9843.049,E2 -9843.049} C_VEL
LIN {X 0,Y 425.282,Z 153.006,A -85,B 0,C 180,E1 -9845.928,E2 -9845.928} C_VEL
LIN {X 0,Y 425.265,Z 153.012,A -85,B 0,C 180,E1 -9849.038,E2 -9849.038} C_VEL
LIN {X 0,Y 425.269,Z 153.015,A -85,B 0,C 180,E1 -9852.654,E2 -9852.654} C_VEL
LIN {X 0,Y 425.261,Z 153.011,A -85,B 0,C 180,E1 -9856.044,E2 -9856.044} C_VEL
LIN {X 0,Y 425.276,Z 153.007,A -85,B 0,C 180,E1 -9859.48,E2 -9859.48} C_VEL
LIN {X 0,Y 425.276,Z 153.012,A -85,B 0,C 180,E1 -9862.489,E2 -9862.489} C_VEL
LIN {X 0,Y 425.307,Z 153.005,A -85,B 0,C 180,E1 -9865.817,E2 -9865.817} C_VEL
LIN {X 0,Y 425.29,Z 153.005,A -85,B 0,C 180,E1 -9869.239,E2 -9869.239} C_VEL
LIN {X 0,Y 425.272,Z 153.01,A -85,B 0,C 180,E1 -9872.437,E2 -9872.437} C_VEL
LIN {X 0,Y 425.347,Z 153.001,A -85,B 0,C 180,E1 -9875.602,E2 -9875.602} C_VEL
LIN {X 0,Y 425.292,Z 153.005,A -85,B 0,C 180,E1 -9878.681,E2 -9878.681} C_VEL
LIN {X 0,Y 425.329,Z 153.007,A -85,B 0,C 180,E1 -9881.703,E2 -9881.703} C_VEL
LIN {X 0,Y 425.347,Z 152.998,A -85,B 0,C 180,E1 -9884.671,E2 -9884.671} C_VEL
LIN {X 0,Y 425.412,Z 152.997,A -85,B 0,C 180,E1 -9887.598,E2 -9887.598} C_VEL
LIN {X 0,Y 425.442,Z 152.993,A -85,B 0,C 180,E1 -9891.45,E2 -9891.45} C_VEL
LIN {X 0,Y 425.55,Z 152.973,A -85,B 0,C 180,E1 -9894.313,E2 -9894.313} C_VEL
LIN {X 0,Y 425.574,Z 152.97,A -85,B 0,C 180,E1 -9898.107,E2 -9898.107} C_VEL
LIN {X 0,Y 425.701,Z 152.954,A -85,B 0,C 180,E1 -9900,E2 -9900} C_VEL
LIN {X 0,Y 425.556,Z 152.976,A -85,B 0,C 180,E1 -9902.84,E2 -9902.84} C_VEL
LIN {X 0,Y 425.499,Z 152.981,A -85,B 0,C 180,E1 -9906.517,E2 -9906.517} C_VEL
LIN {X 0,Y 425.4,Z 152.993,A -85,B 0,C 180,E1 -9909.509,E2 -9909.509} C_VEL
LIN {X 0,Y 425.393,Z 152.999,A -85,B 0,C 180,E1 -9912.904,E2 -9912.904} C_VEL
LIN {X 0,Y 425.362,Z 153.002,A -85,B 0,C 180,E1 -9916.605,E2 -9916.605} C_VEL
LIN {X 0,Y 425.329,Z 153,A -85,B 0,C 180,E1 -9919.636,E2 -9919.636} C_VEL
LIN {X 0,Y 425.307,Z 153.003,A -85,B 0,C 180,E1 -9923.365,E2 -9923.365} C_VEL
LIN {X 0,Y 425.347,Z 153,A -85,B 0,C 180,E1 -9926.844,E2 -9926.844} C_VEL
LIN {X 0,Y 425.291,Z 153.006,A -85,B 0,C 180,E1 -9929.72,E2 -9929.72} C_VEL
LIN {X 0,Y 425.282,Z 153.006,A -85,B 0,C 180,E1 -9933.048,E2 -9933.048} C_VEL
LIN {X 0,Y 425.283,Z 153.01,A -85,B 0,C 180,E1 -9935.929,E2 -9935.929} C_VEL
LIN {X 0,Y 425.294,Z 153.004,A -85,B 0,C 180,E1 -9939.043,E2 -9939.043} C_VEL
LIN {X 0,Y 425.276,Z 153.007,A -85,B 0,C 180,E1 -9942.653,E2 -9942.653} C_VEL
LIN {X 0,Y 425.263,Z 153.013,A -85,B 0,C 180,E1 -9946.044,E2 -9946.044} C_VEL
LIN {X 0,Y 425.275,Z 153.007,A -85,B 0,C 180,E1 -9948.622,E2 -9948.622} C_VEL
LIN {X 0,Y 425.298,Z 153.005,A -85,B 0,C 180,E1 -9951.101,E2 -9951.101} C_VEL
LIN {X 0,Y 425.299,Z 153.004,A -85,B 0,C 180,E1 -9954.664,E2 -9954.664} C_VEL
LIN {X 0,Y 425.266,Z 153.009,A -85,B 0,C 180,E1 -9958.073,E2 -9958.073} C_VEL
LIN {X 0,Y 425.333,Z 153.007,A -85,B 0,C 180,E1 -9961.368,E2 -9961.368} C_VEL
LIN {X 0,Y 425.298,Z 153.007,A -85,B 0,C 180,E1 -9964.555,E2 -9964.555} C_VEL
LIN {X 0,Y 425.357,Z 153.036,A -85,B 0,C 180,E1 -9966.638,E2 -9966.638} C_VEL
LIN {X 0,Y 427.227,Z 163.208,A -85,B 0,C 180,E1 -9969.036,E2 -9969.036} C_VEL
LIN {X 0,Y 426.956,Z 172.415,A -85,B 0,C 180,E1 -9971.041,E2 -9971.041} C_VEL
LIN {X 0,Y 426.861,Z 173.749,A -85,B 0,C 180,E1 -9971.325,E2 -9971.325} C_VEL
LIN {X 0,Y 430.762,Z 194.061,A -85,B 0,C 180,E1 -9971.854,E2 -9971.854} C_VEL
LIN {X 0,Y 429.802,Z 281.542,A -85,B 0,C 180,E1 -9973.342,E2 -9973.342} C_VEL
LIN {X 0,Y 429.378,Z 295.394,A -85,B 0,C 180,E1 -9973.783,E2 -9973.783} C_VEL
LIN {X 0,Y 428.827,Z 307.795,A -85,B 0,C 180,E1 -9974.372,E2 -9974.372} C_VEL
LIN {X 0,Y 428.223,Z 319.649,A -85,B 0,C 180,E1 -9975.141,E2 -9975.141} C_VEL
LIN {X 0,Y 427.566,Z 330.813,A -85,B 0,C 180,E1 -9976.071,E2 -9976.071} C_VEL
LIN {X 0,Y 427.466,Z 333.467,A -85,B 0,C 180,E1 -9976.327,E2 -9976.327} C_VEL
LIN {X 0,Y 426.626,Z 338.187,A -85,B 0,C 180,E1 -9976.799,E2 -9976.799} C_VEL
LIN {X 0,Y 423.316,Z 345.571,A -85,B 0,C 180,E1 -9977.577,E2 -9977.577} C_VEL
LIN {X 0,Y 419.884,Z 352.387,A -85,B 0,C 180,E1 -9978.436,E2 -9978.436} C_VEL
LIN {X 0,Y 418.86,Z 356.231,A -85,B 0,C 180,E1 -9979.025,E2 -9979.025} C_VEL
LIN {X 0,Y 418.319,Z 363.33,A -85,B 0,C 180,E1 -9980.328,E2 -9980.328} C_VEL
LIN {X 0,Y 417.805,Z 369.76,A -85,B 0,C 180,E1 -9981.78,E2 -9981.78} C_VEL
LIN {X 0,Y 417.478,Z 375.154,A -85,B 0,C 180,E1 -9983.332,E2 -9983.332} C_VEL
LIN {X 0,Y 417.321,Z 378.82,A -85,B 0,C 180,E1 -9984.685,E2 -9984.685} C_VEL
LIN {X 0,Y 417.133,Z 381.748,A -85,B 0,C 180,E1 -9986.136,E2 -9986.136} C_VEL
LIN {X 0,Y 417.145,Z 383.15,A -85,B 0,C 180,E1 -9987.103,E2 -9987.103} C_VEL
LIN {X 0,Y 417.015,Z 384.764,A -85,B 0,C 180,E1 -9989.034,E2 -9989.034} C_VEL
LIN {X 0,Y 416.986,Z 384.999,A -85,B 0,C 180,E1 -9990,E2 -9990} C_VEL
LIN {X 0,Y 417.015,Z 384.811,A -85,B 0,C 180,E1 -9990.966,E2 -9990.966} C_VEL
LIN {X 0,Y 417.144,Z 383.258,A -85,B 0,C 180,E1 -9992.897,E2 -9992.897} C_VEL
LIN {X 0,Y 417.128,Z 381.903,A -85,B 0,C 180,E1 -9993.864,E2 -9993.864} C_VEL
LIN {X 0,Y 417.31,Z 379.034,A -85,B 0,C 180,E1 -9995.315,E2 -9995.315} C_VEL
LIN {X 0,Y 417.479,Z 375.146,A -85,B 0,C 180,E1 -9996.767,E2 -9996.767} C_VEL
LIN {X 0,Y 417.791,Z 370.129,A -85,B 0,C 180,E1 -9998.221,E2 -9998.221} C_VEL
LIN {X 0,Y 418.296,Z 363.813,A -85,B 0,C 180,E1 -9999.672,E2 -9999.672} C_VEL
LIN {X 0,Y 418.834,Z 355.907,A -85,B 0,C 180,E1 -10001.126,E2 -10001.126} C_VEL
LIN {X 0,Y 419.485,Z 347.846,A -85,B 0,C 180,E1 -10002.334,E2 -10002.334} C_VEL
LIN {X 0,Y 420.28,Z 338.008,A -85,B 0,C 180,E1 -10003.539,E2 -10003.539} C_VEL
LIN {X 0,Y 420.948,Z 326.949,A -85,B 0,C 180,E1 -10004.627,E2 -10004.627} C_VEL
LIN {X 0,Y 421.6,Z 316.103,A -85,B 0,C 180,E1 -10005.469,E2 -10005.469} C_VEL
LIN {X 0,Y 422.27,Z 304.124,A -85,B 0,C 180,E1 -10006.187,E2 -10006.187} C_VEL
LIN {X 0,Y 422.748,Z 291.855,A -85,B 0,C 180,E1 -10006.727,E2 -10006.727} C_VEL
LIN {X 0,Y 423.127,Z 279.239,A -85,B 0,C 180,E1 -10007.084,E2 -10007.084} C_VEL
LIN {X 0,Y 423.95,Z 193.958,A -85,B 0,C 180,E1 -10008.55,E2 -10008.55} C_VEL
LIN {X 0,Y 419.967,Z 173.81,A -85,B 0,C 180,E1 -10009.113,E2 -10009.113} C_VEL
LIN {X 0,Y 420.366,Z 164.933,A -85,B 0,C 180,E1 -10011.066,E2 -10011.066} C_VEL
LIN {X 0,Y 418.309,Z 153.879,A -85,B 0,C 180,E1 -10013.714,E2 -10013.714} C_VEL
LIN {X 0,Y 418.312,Z 153.878,A -85,B 0,C 180,E1 -10017.07,E2 -10017.07} C_VEL
LIN {X 0,Y 418.246,Z 153.886,A -85,B 0,C 180,E1 -10020.272,E2 -10020.272} C_VEL
LIN {X 0,Y 418.248,Z 153.882,A -85,B 0,C 180,E1 -10023.677,E2 -10023.677} C_VEL
LIN {X 0,Y 418.24,Z 153.883,A -85,B 0,C 180,E1 -10027.224,E2 -10027.224} C_VEL
LIN {X 0,Y 418.245,Z 153.883,A -85,B 0,C 180,E1 -10029.682,E2 -10029.682} C_VEL
LIN {X 0,Y 418.231,Z 153.891,A -85,B 0,C 180,E1 -10032.321,E2 -10032.321} C_VEL
LIN {X 0,Y 418.238,Z 153.884,A -85,B 0,C 180,E1 -10035.109,E2 -10035.109} C_VEL
LIN {X 0,Y 418.241,Z 153.886,A -85,B 0,C 180,E1 -10037.767,E2 -10037.767} C_VEL
LIN {X 0,Y 418.253,Z 153.883,A -85,B 0,C 180,E1 -10040.619,E2 -10040.619} C_VEL
LIN {X 0,Y 418.243,Z 153.889,A -85,B 0,C 180,E1 -10043.976,E2 -10043.976} C_VEL
LIN {X 0,Y 418.257,Z 153.882,A -85,B 0,C 180,E1 -10047.156,E2 -10047.156} C_VEL
LIN {X 0,Y 418.268,Z 153.88,A -85,B 0,C 180,E1 -10050.895,E2 -10050.895} C_VEL
LIN {X 0,Y 418.27,Z 153.881,A -85,B 0,C 180,E1 -10054.096,E2 -10054.096} C_VEL
LIN {X 0,Y 418.238,Z 153.888,A -85,B 0,C 180,E1 -10057.264,E2 -10057.264} C_VEL
LIN {X 0,Y 418.283,Z 153.878,A -85,B 0,C 180,E1 -10060.364,E2 -10060.364} C_VEL
LIN {X 0,Y 418.317,Z 153.88,A -85,B 0,C 180,E1 -10063.404,E2 -10063.404} C_VEL
LIN {X 0,Y 418.346,Z 153.875,A -85,B 0,C 180,E1 -10066.999,E2 -10066.999} C_VEL
LIN {X 0,Y 418.34,Z 153.871,A -85,B 0,C 180,E1 -10070.329,E2 -10070.329} C_VEL
LIN {X 0,Y 418.486,Z 153.857,A -85,B 0,C 180,E1 -10073.249,E2 -10073.249} C_VEL
LIN {X 0,Y 418.338,Z 153.876,A -85,B 0,C 180,E1 -10075.181,E2 -10075.181} C_VEL
LIN {X 0,Y 418.544,Z 153.846,A -85,B 0,C 180,E1 -10078.075,E2 -10078.075} C_VEL
LIN {X 0,Y 418.67,Z 153.83,A -85,B 0,C 180,E1 -10080,E2 -10080} C_VEL
LIN {X 0,Y 418.508,Z 153.855,A -85,B 0,C 180,E1 -10082.888,E2 -10082.888} C_VEL
LIN {X 0,Y 418.486,Z 153.858,A -85,B 0,C 180,E1 -10086.751,E2 -10086.751} C_VEL
LIN {X 0,Y 418.339,Z 153.871,A -85,B 0,C 180,E1 -10089.671,E2 -10089.671} C_VEL
LIN {X 0,Y 418.345,Z 153.871,A -85,B 0,C 180,E1 -10093.001,E2 -10093.001} C_VEL
LIN {X 0,Y 418.311,Z 153.877,A -85,B 0,C 180,E1 -10096.735,E2 -10096.735} C_VEL
LIN {X 0,Y 418.269,Z 153.882,A -85,B 0,C 180,E1 -10099.79,E2 -10099.79} C_VEL
LIN {X 0,Y 418.231,Z 153.886,A -85,B 0,C 180,E1 -10102.737,E2 -10102.737} C_VEL
LIN {X 0,Y 418.267,Z 153.886,A -85,B 0,C 180,E1 -10105.904,E2 -10105.904} C_VEL
LIN {X 0,Y 418.264,Z 153.881,A -85,B 0,C 180,E1 -10109.162,E2 -10109.162} C_VEL
LIN {X 0,Y 418.257,Z 153.881,A -85,B 0,C 180,E1 -10112.844,E2 -10112.844} C_VEL
LIN {X 0,Y 418.243,Z 153.885,A -85,B 0,C 180,E1 -10116.238,E2 -10116.238} C_VEL
LIN {X 0,Y 418.241,Z 153.889,A -85,B 0,C 180,E1 -10119.683,E2 -10119.683} C_VEL
LIN {X 0,Y 418.223,Z 153.886,A -85,B 0,C 180,E1 -10122.32,E2 -10122.32} C_VEL
LIN {X 0,Y 418.235,Z 153.887,A -85,B 0,C 180,E1 -10125.109,E2 -10125.109} C_VEL
LIN {X 0,Y 418.232,Z 153.887,A -85,B 0,C 180,E1 -10127.766,E2 -10127.766} C_VEL
LIN {X 0,Y 418.24,Z 153.887,A -85,B 0,C 180,E1 -10131.557,E2 -10131.557} C_VEL
LIN {X 0,Y 418.258,Z 153.888,A -85,B 0,C 180,E1 -10135.159,E2 -10135.159} C_VEL
LIN {X 0,Y 418.245,Z 153.885,A -85,B 0,C 180,E1 -10137.472,E2 -10137.472} C_VEL
LIN {X 0,Y 418.262,Z 153.888,A -85,B 0,C 180,E1 -10140.898,E2 -10140.898} C_VEL
LIN {X 0,Y 418.259,Z 153.989,A -85,B 0,C 180,E1 -10142.987,E2 -10142.987} C_VEL
LIN {X 0,Y 420.81,Z 166.732,A -85,B 0,C 180,E1 -10145.847,E2 -10145.847} C_VEL
LIN {X 0,Y 421.063,Z 170.45,A -85,B 0,C 180,E1 -10146.637,E2 -10146.637} C_VEL
LIN {X 0,Y 419.923,Z 188.061,A -85,B 0,C 180,E1 -10150.211,E2 -10150.211} C_VEL
LIN {X 0,Y 419.715,Z 191.537,A -85,B 0,C 180,E1 -10150.911,E2 -10150.911} C_VEL
LIN {X 0,Y 423.72,Z 216.043,A -85,B 0,C 180,E1 -10151.55,E2 -10151.55} C_VEL
LIN {X 0,Y 422.916,Z 299.841,A -85,B 0,C 180,E1 -10153,E2 -10153} C_VEL
LIN {X 0,Y 422.428,Z 312.312,A -85,B 0,C 180,E1 -10153.384,E2 -10153.384} C_VEL
LIN {X 0,Y 421.803,Z 325.217,A -85,B 0,C 180,E1 -10153.981,E2 -10153.981} C_VEL
LIN {X 0,Y 421.049,Z 337.469,A -85,B 0,C 180,E1 -10154.758,E2 -10154.758} C_VEL
